LIN {X 0,Y 469.411,Z 470.46,A -85,B 0,C 180,E1 -7614.274,E2 -7614.274} C_VEL
LIN {X 0,Y 468.875,Z 476.006,A -85,B 0,C 180,E1 -7617.076,E2 -7617.076} C_VEL
LIN {X 0,Y 468.362,Z 482.236,A -85,B 0,C 180,E1 -7619.822,E2 -7619.822} C_VEL
LIN {X 0,Y 467.901,Z 490.724,A -85,B 0,C 180,E1 -7623.217,E2 -7623.217} C_VEL
LIN {X 0,Y 467.584,Z 498.381,A -85,B 0,C 180,E1 -7626.057,E2 -7626.057} C_VEL
LIN {X 0,Y 467.333,Z 507.548,A -85,B 0,C 180,E1 -7629.304,E2 -7629.304} C_VEL
LIN {X 0,Y 467.075,Z 516.898,A -85,B 0,C 180,E1 -7632.486,E2 -7632.486} C_VEL
LIN {X 0,Y 467.02,Z 523.224,A -85,B 0,C 180,E1 -7634.591,E2 -7634.591} C_VEL
LIN {X 0,Y 468.953,Z 538.487,A -85,B 0,C 180,E1 -7635.113,E2 -7635.113} C_VEL
LIN {X 0,Y 469.751,Z 545.686,A -85,B 0,C 180,E1 -7635.432,E2 -7635.432} C_VEL
LIN {X 0,Y 469.303,Z 557.555,A -85,B 0,C 180,E1 -7636.026,E2 -7636.026} C_VEL
LIN {X 0,Y 468.855,Z 569.316,A -85,B 0,C 180,E1 -7636.786,E2 -7636.786} C_VEL
LIN {X 0,Y 468.371,Z 580.525,A -85,B 0,C 180,E1 -7637.703,E2 -7637.703} C_VEL
LIN {X 0,Y 467.91,Z 590.813,A -85,B 0,C 180,E1 -7638.74,E2 -7638.74} C_VEL
LIN {X 0,Y 467.467,Z 599.647,A -85,B 0,C 180,E1 -7639.825,E2 -7639.825} C_VEL
LIN {X 0,Y 467.142,Z 608.26,A -85,B 0,C 180,E1 -7641.129,E2 -7641.129} C_VEL
LIN {X 0,Y 466.928,Z 615.206,A -85,B 0,C 180,E1 -7642.432,E2 -7642.432} C_VEL
LIN {X 0,Y 466.769,Z 621.589,A -85,B 0,C 180,E1 -7643.95,E2 -7643.95} C_VEL
LIN {X 0,Y 466.701,Z 625.734,A -85,B 0,C 180,E1 -7645.249,E2 -7645.249} C_VEL
LIN {X 0,Y 466.73,Z 628.807,A -85,B 0,C 180,E1 -7646.547,E2 -7646.547} C_VEL
LIN {X 0,Y 466.71,Z 630.278,A -85,B 0,C 180,E1 -7647.411,E2 -7647.411} C_VEL
LIN {X 0,Y 466.694,Z 631.332,A -85,B 0,C 180,E1 -7648.274,E2 -7648.274} C_VEL
LIN {X 0,Y 466.62,Z 631.982,A -85,B 0,C 180,E1 -7649.137,E2 -7649.137} C_VEL
LIN {X 0,Y 466.598,Z 632.228,A -85,B 0,C 180,E1 -7650,E2 -7650} C_VEL
LIN {X 0,Y 466.693,Z 631.43,A -85,B 0,C 180,E1 -7651.726,E2 -7651.726} C_VEL
LIN {X 0,Y 466.7,Z 630.431,A -85,B 0,C 180,E1 -7652.589,E2 -7652.589} C_VEL
LIN {X 0,Y 466.73,Z 629.01,A -85,B 0,C 180,E1 -7653.453,E2 -7653.453} C_VEL
LIN {X 0,Y 466.701,Z 626.022,A -85,B 0,C 180,E1 -7654.751,E2 -7654.751} C_VEL
LIN {X 0,Y 466.768,Z 621.97,A -85,B 0,C 180,E1 -7656.05,E2 -7656.05} C_VEL
LIN {X 0,Y 466.928,Z 615.723,A -85,B 0,C 180,E1 -7657.568,E2 -7657.568} C_VEL
LIN {X 0,Y 467.163,Z 608.913,A -85,B 0,C 180,E1 -7658.87,E2 -7658.87} C_VEL
LIN {X 0,Y 467.485,Z 600.458,A -85,B 0,C 180,E1 -7660.174,E2 -7660.174} C_VEL
LIN {X 0,Y 467.928,Z 591.764,A -85,B 0,C 180,E1 -7661.259,E2 -7661.259} C_VEL
LIN {X 0,Y 468.375,Z 581.539,A -85,B 0,C 180,E1 -7662.305,E2 -7662.305} C_VEL
LIN {X 0,Y 468.887,Z 570.553,A -85,B 0,C 180,E1 -7663.213,E2 -7663.213} C_VEL
LIN {X 0,Y 469.389,Z 558.907,A -85,B 0,C 180,E1 -7663.971,E2 -7663.971} C_VEL
LIN {X 0,Y 469.901,Z 545.767,A -85,B 0,C 180,E1 -7664.619,E2 -7664.619} C_VEL
LIN {X 0,Y 468.192,Z 532.419,A -85,B 0,C 180,E1 -7665.144,E2 -7665.144} C_VEL
LIN {X 0,Y 467.098,Z 524.822,A -85,B 0,C 180,E1 -7665.381,E2 -7665.381} C_VEL
LIN {X 0,Y 467.284,Z 515.355,A -85,B 0,C 180,E1 -7668.643,E2 -7668.643} C_VEL
LIN {X 0,Y 467.574,Z 505.589,A -85,B 0,C 180,E1 -7672.072,E2 -7672.072} C_VEL
LIN {X 0,Y 467.924,Z 496.629,A -85,B 0,C 180,E1 -7675.285,E2 -7675.285} C_VEL
LIN {X 0,Y 468.323,Z 488.674,A -85,B 0,C 180,E1 -7678.21,E2 -7678.21} C_VEL
LIN {X 0,Y 468.742,Z 480.586,A -85,B 0,C 180,E1 -7681.282,E2 -7681.282} C_VEL
LIN {X 0,Y 469.161,Z 473.387,A -85,B 0,C 180,E1 -7684.097,E2 -7684.097} C_VEL
LIN {X 0,Y 469.33,Z 468.592,A -85,B 0,C 180,E1 -7686.038,E2 -7686.038} C_VEL
LIN {X 0,Y 468.349,Z 462.399,A -85,B 0,C 180,E1 -7688.711,E2 -7688.711} C_VEL
LIN {X 0,Y 467.578,Z 458.244,A -85,B 0,C 180,E1 -7690.618,E2 -7690.618} C_VEL
LIN {X 0,Y 467.558,Z 458.244,A -85,B 0,C 180,E1 -7693.744,E2 -7693.744} C_VEL
LIN {X 0,Y 467.579,Z 458.244,A -85,B 0,C 180,E1 -7696.258,E2 -7696.258} C_VEL
LIN {X 0,Y 467.585,Z 458.241,A -85,B 0,C 180,E1 -7698.722,E2 -7698.722} C_VEL
LIN {X 0,Y 467.566,Z 458.242,A -85,B 0,C 180,E1 -7701.956,E2 -7701.956} C_VEL
LIN {X 0,Y 467.566,Z 458.245,A -85,B 0,C 180,E1 -7705.167,E2 -7705.167} C_VEL
LIN {X 0,Y 467.584,Z 458.241,A -85,B 0,C 180,E1 -7708.26,E2 -7708.26} C_VEL
LIN {X 0,Y 467.579,Z 458.243,A -85,B 0,C 180,E1 -7711.251,E2 -7711.251} C_VEL
LIN {X 0,Y 467.618,Z 458.238,A -85,B 0,C 180,E1 -7713.2,E2 -7713.2} C_VEL
LIN {X 0,Y 467.593,Z 458.243,A -85,B 0,C 180,E1 -7716.468,E2 -7716.468} C_VEL
LIN {X 0,Y 467.626,Z 458.236,A -85,B 0,C 180,E1 -7719.777,E2 -7719.777} C_VEL
LIN {X 0,Y 467.611,Z 458.24,A -85,B 0,C 180,E1 -7722.507,E2 -7722.507} C_VEL
LIN {X 0,Y 467.609,Z 458.238,A -85,B 0,C 180,E1 -7725.197,E2 -7725.197} C_VEL
LIN {X 0,Y 467.658,Z 458.232,A -85,B 0,C 180,E1 -7727.855,E2 -7727.855} C_VEL
LIN {X 0,Y 467.683,Z 458.228,A -85,B 0,C 180,E1 -7731.357,E2 -7731.357} C_VEL
LIN {X 0,Y 467.746,Z 458.222,A -85,B 0,C 180,E1 -7733.963,E2 -7733.963} C_VEL
LIN {X 0,Y 467.861,Z 458.204,A -85,B 0,C 180,E1 -7737.417,E2 -7737.417} C_VEL
LIN {X 0,Y 467.885,Z 458.206,A -85,B 0,C 180,E1 -7740,E2 -7740} C_VEL
LIN {X 0,Y 467.861,Z 458.208,A -85,B 0,C 180,E1 -7742.583,E2 -7742.583} C_VEL
LIN {X 0,Y 467.746,Z 458.223,A -85,B 0,C 180,E1 -7746.038,E2 -7746.038} C_VEL
LIN {X 0,Y 467.684,Z 458.229,A -85,B 0,C 180,E1 -7748.643,E2 -7748.643} C_VEL
LIN {X 0,Y 467.658,Z 458.233,A -85,B 0,C 180,E1 -7752.146,E2 -7752.146} C_VEL
LIN {X 0,Y 467.642,Z 458.235,A -85,B 0,C 180,E1 -7755.695,E2 -7755.695} C_VEL
LIN {X 0,Y 467.62,Z 458.236,A -85,B 0,C 180,E1 -7758.765,E2 -7758.765} C_VEL
LIN {X 0,Y 467.583,Z 458.241,A -85,B 0,C 180,E1 -7761.268,E2 -7761.268} C_VEL
LIN {X 0,Y 467.574,Z 458.242,A -85,B 0,C 180,E1 -7763.943,E2 -7763.943} C_VEL
LIN {X 0,Y 467.619,Z 458.236,A -85,B 0,C 180,E1 -7766.8,E2 -7766.8} C_VEL
LIN {X 0,Y 467.557,Z 458.246,A -85,B 0,C 180,E1 -7769.738,E2 -7769.738} C_VEL
LIN {X 0,Y 467.586,Z 458.24,A -85,B 0,C 180,E1 -7772.759,E2 -7772.759} C_VEL
LIN {X 0,Y 467.559,Z 458.247,A -85,B 0,C 180,E1 -7775.89,E2 -7775.89} C_VEL
LIN {X 0,Y 467.579,Z 458.241,A -85,B 0,C 180,E1 -7779.146,E2 -7779.146} C_VEL
LIN {X 0,Y 467.589,Z 458.24,A -85,B 0,C 180,E1 -7782.567,E2 -7782.567} C_VEL
LIN {X 0,Y 467.574,Z 458.243,A -85,B 0,C 180,E1 -7785.053,E2 -7785.053} C_VEL
LIN {X 0,Y 467.592,Z 458.238,A -85,B 0,C 180,E1 -7787.44,E2 -7787.44} C_VEL
LIN {X 0,Y 467.586,Z 458.242,A -85,B 0,C 180,E1 -7790.856,E2 -7790.856} C_VEL
LIN {X 0,Y 467.566,Z 458.246,A -85,B 0,C 180,E1 -7794.261,E2 -7794.261} C_VEL
LIN {X 0,Y 467.585,Z 458.241,A -85,B 0,C 180,E1 -7797.321,E2 -7797.321} C_VEL
LIN {X 0,Y 467.574,Z 458.243,A -85,B 0,C 180,E1 -7800.668,E2 -7800.668} C_VEL
LIN {X 0,Y 467.62,Z 458.235,A -85,B 0,C 180,E1 -7803.2,E2 -7803.2} C_VEL
LIN {X 0,Y 467.597,Z 458.241,A -85,B 0,C 180,E1 -7806.468,E2 -7806.468} C_VEL
LIN {X 0,Y 467.627,Z 458.236,A -85,B 0,C 180,E1 -7809.777,E2 -7809.777} C_VEL
LIN {X 0,Y 467.603,Z 458.239,A -85,B 0,C 180,E1 -7812.507,E2 -7812.507} C_VEL
LIN {X 0,Y 467.611,Z 458.237,A -85,B 0,C 180,E1 -7815.197,E2 -7815.197} C_VEL
LIN {X 0,Y 467.602,Z 458.238,A -85,B 0,C 180,E1 -7815.421,E2 -7815.421} C_VEL
LIN {X 0,Y 466.931,Z 458.326,A -85,B 0,C 180,E1 -7816.14,E2 -7816.14} C_VEL
LIN {X 0,Y 464.088,Z 458.675,A -85,B 0,C 180,E1 -7817.309,E2 -7817.309} C_VEL
LIN {X 0,Y 461.689,Z 458.975,A -85,B 0,C 180,E1 -7818.251,E2 -7818.251} C_VEL
LIN {X 0,Y 460.662,Z 459.103,A -85,B 0,C 180,E1 -7818.979,E2 -7818.979} C_VEL
LIN {X 0,Y 460.58,Z 459.113,A -85,B 0,C 180,E1 -7819.225,E2 -7819.225} C_VEL
LIN {X 0,Y 460.673,Z 459.102,A -85,B 0,C 180,E1 -7822.588,E2 -7822.588} C_VEL
LIN {X 0,Y 460.694,Z 459.098,A -85,B 0,C 180,E1 -7824.748,E2 -7824.748} C_VEL
LIN {X 0,Y 460.805,Z 459.087,A -85,B 0,C 180,E1 -7827.378,E2 -7827.378} C_VEL
LIN {X 0,Y 460.858,Z 459.081,A -85,B 0,C 180,E1 -7830,E2 -7830} C_VEL
LIN {X 0,Y 460.805,Z 459.084,A -85,B 0,C 180,E1 -7832.623,E2 -7832.623} C_VEL
LIN {X 0,Y 460.712,Z 459.099,A -85,B 0,C 180,E1 -7836.13,E2 -7836.13} C_VEL
LIN {X 0,Y 460.626,Z 459.106,A -85,B 0,C 180,E1 -7838.776,E2 -7838.776} C_VEL
LIN {X 0,Y 460.618,Z 459.111,A -85,B 0,C 180,E1 -7842.445,E2 -7842.445} C_VEL
LIN {X 0,Y 460.605,Z 459.112,A -85,B 0,C 180,E1 -7845.998,E2 -7845.998} C_VEL
LIN {X 0,Y 460.576,Z 459.114,A -85,B 0,C 180,E1 -7848.902,E2 -7848.902} C_VEL
LIN {X 0,Y 460.521,Z 459.12,A -85,B 0,C 180,E1 -7851.486,E2 -7851.486} C_VEL
LIN {X 0,Y 460.547,Z 459.117,A -85,B 0,C 180,E1 -7854.332,E2 -7854.332} C_VEL
LIN {X 0,Y 460.578,Z 459.114,A -85,B 0,C 180,E1 -7857.244,E2 -7857.244} C_VEL
LIN {X 0,Y 460.515,Z 459.121,A -85,B 0,C 180,E1 -7860.24,E2 -7860.24} C_VEL
LIN {X 0,Y 460.533,Z 459.121,A -85,B 0,C 180,E1 -7863.325,E2 -7863.325} C_VEL
LIN {X 0,Y 460.481,Z 459.124,A -85,B 0,C 180,E1 -7866.529,E2 -7866.529} C_VEL
LIN {X 0,Y 460.549,Z 459.117,A -85,B 0,C 180,E1 -7868.898,E2 -7868.898} C_VEL
LIN {X 0,Y 460.527,Z 459.122,A -85,B 0,C 180,E1 -7872.181,E2 -7872.181} C_VEL
LIN {X 0,Y 460.518,Z 459.122,A -85,B 0,C 180,E1 -7875.411,E2 -7875.411} C_VEL
LIN {X 0,Y 460.536,Z 459.12,A -85,B 0,C 180,E1 -7878.397,E2 -7878.397} C_VEL
LIN {X 0,Y 460.529,Z 459.119,A -85,B 0,C 180,E1 -7881.267,E2 -7881.267} C_VEL
LIN {X 0,Y 460.438,Z 459.132,A -85,B 0,C 180,E1 -7884.548,E2 -7884.548} C_VEL
LIN {X 0,Y 460.116,Z 459.175,A -85,B 0,C 180,E1 -7887.683,E2 -7887.683} C_VEL
LIN {X 0,Y 459.914,Z 459.335,A -85,B 0,C 180,E1 -7889.716,E2 -7889.716} C_VEL
LIN {X 0,Y 459.916,Z 462.429,A -85,B 0,C 180,E1 -7892.714,E2 -7892.714} C_VEL
LIN {X 0,Y 459.808,Z 465.5,A -85,B 0,C 180,E1 -7895.626,E2 -7895.626} C_VEL
LIN {X 0,Y 459.763,Z 468.905,A -85,B 0,C 180,E1 -7898.821,E2 -7898.821} C_VEL
LIN {X 0,Y 459.71,Z 472.578,A -85,B 0,C 180,E1 -7902.196,E2 -7902.196} C_VEL
LIN {X 0,Y 459.717,Z 475.164,A -85,B 0,C 180,E1 -7904.538,E2 -7904.538} C_VEL
LIN {X 0,Y 462.865,Z 489.688,A -85,B 0,C 180,E1 -7905.125,E2 -7905.125} C_VEL
LIN {X 0,Y 463.135,Z 494.215,A -85,B 0,C 180,E1 -7905.331,E2 -7905.331} C_VEL
LIN {X 0,Y 462.75,Z 505.895,A -85,B 0,C 180,E1 -7905.936,E2 -7905.936} C_VEL
LIN {X 0,Y 462.3,Z 517.223,A -85,B 0,C 180,E1 -7906.696,E2 -7906.696} C_VEL
LIN {X 0,Y 461.794,Z 528.968,A -85,B 0,C 180,E1 -7907.698,E2 -7907.698} C_VEL
LIN {X 0,Y 461.227,Z 539.33,A -85,B 0,C 180,E1 -7908.797,E2 -7908.797} C_VEL
LIN {X 0,Y 460.77,Z 549.23,A -85,B 0,C 180,E1 -7910.119,E2 -7910.119} C_VEL
LIN {X 0,Y 460.392,Z 557.21,A -85,B 0,C 180,E1 -7911.44,E2 -7911.44} C_VEL
LIN {X 0,Y 460.132,Z 562.609,A -85,B 0,C 180,E1 -7912.54,E2 -7912.54} C_VEL
LIN {X 0,Y 460.009,Z 567.893,A -85,B 0,C 180,E1 -7913.861,E2 -7913.861} C_VEL
LIN {X 0,Y 459.791,Z 572.006,A -85,B 0,C 180,E1 -7915.177,E2 -7915.177} C_VEL
LIN {X 0,Y 459.725,Z 575.053,A -85,B 0,C 180,E1 -7916.494,E2 -7916.494} C_VEL
LIN {X 0,Y 459.705,Z 576.536,A -85,B 0,C 180,E1 -7917.371,E2 -7917.371} C_VEL
LIN {X 0,Y 459.636,Z 577.592,A -85,B 0,C 180,E1 -7918.247,E2 -7918.247} C_VEL
LIN {X 0,Y 459.531,Z 578.546,A -85,B 0,C 180,E1 -7920,E2 -7920} C_VEL
LIN {X 0,Y 459.554,Z 578.388,A -85,B 0,C 180,E1 -7920.876,E2 -7920.876} C_VEL
LIN {X 0,Y 459.736,Z 576.871,A -85,B 0,C 180,E1 -7922.628,E2 -7922.628} C_VEL
LIN {X 0,Y 459.733,Z 575.522,A -85,B 0,C 180,E1 -7923.506,E2 -7923.506} C_VEL
LIN {X 0,Y 459.809,Z 572.652,A -85,B 0,C 180,E1 -7924.822,E2 -7924.822} C_VEL
LIN {X 0,Y 460.009,Z 568.73,A -85,B 0,C 180,E1 -7926.139,E2 -7926.139} C_VEL
LIN {X 0,Y 460.179,Z 563.651,A -85,B 0,C 180,E1 -7927.459,E2 -7927.459} C_VEL
LIN {X 0,Y 460.493,Z 557.247,A -85,B 0,C 180,E1 -7928.779,E2 -7928.779} C_VEL
LIN {X 0,Y 460.885,Z 549.276,A -85,B 0,C 180,E1 -7930.1,E2 -7930.1} C_VEL
LIN {X 0,Y 461.301,Z 541.139,A -85,B 0,C 180,E1 -7931.201,E2 -7931.201} C_VEL
LIN {X 0,Y 461.9,Z 531.186,A -85,B 0,C 180,E1 -7932.299,E2 -7932.299} C_VEL
LIN {X 0,Y 462.345,Z 519.856,A -85,B 0,C 180,E1 -7933.304,E2 -7933.304} C_VEL
LIN {X 0,Y 462.828,Z 509.159,A -85,B 0,C 180,E1 -7934.061,E2 -7934.061} C_VEL
LIN {X 0,Y 463.277,Z 497.241,A -85,B 0,C 180,E1 -7934.72,E2 -7934.72} C_VEL
LIN {X 0,Y 463.399,Z 492.393,A -85,B 0,C 180,E1 -7934.941,E2 -7934.941} C_VEL
LIN {X 0,Y 461.369,Z 482.734,A -85,B 0,C 180,E1 -7935.391,E2 -7935.391} C_VEL
LIN {X 0,Y 459.919,Z 477.276,A -85,B 0,C 180,E1 -7935.64,E2 -7935.64} C_VEL
LIN {X 0,Y 460.006,Z 474.424,A -85,B 0,C 180,E1 -7938.714,E2 -7938.714} C_VEL
LIN {X 0,Y 460.053,Z 471.957,A -85,B 0,C 180,E1 -7941.508,E2 -7941.508} C_VEL
LIN {X 0,Y 460.187,Z 469.59,A -85,B 0,C 180,E1 -7944.352,E2 -7944.352} C_VEL
LIN {X 0,Y 460.415,Z 466.954,A -85,B 0,C 180,E1 -7947.706,E2 -7947.706} C_VEL
LIN {X 0,Y 460.609,Z 464.479,A -85,B 0,C 180,E1 -7951.3,E2 -7951.3} C_VEL
LIN {X 0,Y 460.817,Z 462.698,A -85,B 0,C 180,E1 -7954.353,E2 -7954.353} C_VEL
LIN {X 0,Y 460.839,Z 461.746,A -85,B 0,C 180,E1 -7956.496,E2 -7956.496} C_VEL
LIN {X 0,Y 460.839,Z 461.064,A -85,B 0,C 180,E1 -7958.942,E2 -7958.942} C_VEL
LIN {X 0,Y 460.826,Z 460.856,A -85,B 0,C 180,E1 -7961.643,E2 -7961.643} C_VEL
LIN {X 0,Y 460.959,Z 461.487,A -85,B 0,C 180,E1 -7964.535,E2 -7964.535} C_VEL
LIN {X 0,Y 461.186,Z 462.915,A -85,B 0,C 180,E1 -7967.01,E2 -7967.01} C_VEL
LIN {X 0,Y 461.639,Z 465.205,A -85,B 0,C 180,E1 -7969.57,E2 -7969.57} C_VEL
LIN {X 0,Y 462.201,Z 468.615,A -85,B 0,C 180,E1 -7972.25,E2 -7972.25} C_VEL
LIN {X 0,Y 462.403,Z 470.846,A -85,B 0,C 180,E1 -7973.663,E2 -7973.663} C_VEL
LIN {X 0,Y 462.167,Z 474.66,A -85,B 0,C 180,E1 -7975.761,E2 -7975.761} C_VEL
LIN {X 0,Y 461.523,Z 481.094,A -85,B 0,C 180,E1 -7978.819,E2 -7978.819} C_VEL
LIN {X 0,Y 461.005,Z 489.008,A -85,B 0,C 180,E1 -7982.154,E2 -7982.154} C_VEL
LIN {X 0,Y 460.615,Z 496.842,A -85,B 0,C 180,E1 -7985.191,E2 -7985.191} C_VEL
LIN {X 0,Y 460.323,Z 505.906,A -85,B 0,C 180,E1 -7988.505,E2 -7988.505} C_VEL
LIN {X 0,Y 460.059,Z 515.164,A -85,B 0,C 180,E1 -7991.75,E2 -7991.75} C_VEL
LIN {X 0,Y 459.944,Z 522.743,A -85,B 0,C 180,E1 -7994.336,E2 -7994.336} C_VEL
LIN {X 0,Y 461.694,Z 536.071,A -85,B 0,C 180,E1 -7994.79,E2 -7994.79} C_VEL
LIN {X 0,Y 462.832,Z 546.609,A -85,B 0,C 180,E1 -7995.265,E2 -7995.265} C_VEL
LIN {X 0,Y 462.324,Z 559.032,A -85,B 0,C 180,E1 -7995.923,E2 -7995.923} C_VEL
LIN {X 0,Y 461.735,Z 571.691,A -85,B 0,C 180,E1 -7996.802,E2 -7996.802} C_VEL
LIN {X 0,Y 461.195,Z 583.009,A -85,B 0,C 180,E1 -7997.793,E2 -7997.793} C_VEL
LIN {X 0,Y 460.783,Z 592.205,A -85,B 0,C 180,E1 -7998.786,E2 -7998.786} C_VEL
LIN {X 0,Y 460.297,Z 602.22,A -85,B 0,C 180,E1 -8000.109,E2 -8000.109} C_VEL
LIN {X 0,Y 460.03,Z 610.282,A -85,B 0,C 180,E1 -8001.434,E2 -8001.434} C_VEL
LIN {X 0,Y 459.775,Z 617.67,A -85,B 0,C 180,E1 -8002.976,E2 -8002.976} C_VEL
LIN {X 0,Y 459.683,Z 622.616,A -85,B 0,C 180,E1 -8004.297,E2 -8004.297} C_VEL
LIN {X 0,Y 459.587,Z 626.407,A -85,B 0,C 180,E1 -8005.615,E2 -8005.615} C_VEL
LIN {X 0,Y 459.643,Z 628.375,A -85,B 0,C 180,E1 -8006.493,E2 -8006.493} C_VEL
LIN {X 0,Y 459.63,Z 629.853,A -85,B 0,C 180,E1 -8007.371,E2 -8007.371} C_VEL
LIN {X 0,Y 459.631,Z 630.914,A -85,B 0,C 180,E1 -8008.247,E2 -8008.247} C_VEL
LIN {X 0,Y 459.553,Z 631.57,A -85,B 0,C 180,E1 -8009.124,E2 -8009.124} C_VEL
LIN {X 0,Y 459.53,Z 631.819,A -85,B 0,C 180,E1 -8010,E2 -8010} C_VEL
LIN {X 0,Y 459.553,Z 631.62,A -85,B 0,C 180,E1 -8010.876,E2 -8010.876} C_VEL
LIN {X 0,Y 459.63,Z 631.024,A -85,B 0,C 180,E1 -8011.752,E2 -8011.752} C_VEL
LIN {X 0,Y 459.621,Z 630.022,A -85,B 0,C 180,E1 -8012.629,E2 -8012.629} C_VEL
LIN {X 0,Y 459.627,Z 628.595,A -85,B 0,C 180,E1 -8013.506,E2 -8013.506} C_VEL
LIN {X 0,Y 459.631,Z 625.603,A -85,B 0,C 180,E1 -8014.824,E2 -8014.824} C_VEL
LIN {X 0,Y 459.714,Z 620.477,A -85,B 0,C 180,E1 -8016.431,E2 -8016.431} C_VEL
LIN {X 0,Y 459.896,Z 614.255,A -85,B 0,C 180,E1 -8017.905,E2 -8017.905} C_VEL
LIN {X 0,Y 460.185,Z 607.179,A -85,B 0,C 180,E1 -8019.228,E2 -8019.228} C_VEL
LIN {X 0,Y 460.537,Z 598.326,A -85,B 0,C 180,E1 -8020.552,E2 -8020.552} C_VEL
LIN {X 0,Y 461.115,Z 588.309,A -85,B 0,C 180,E1 -8021.762,E2 -8021.762} C_VEL
LIN {X 0,Y 461.583,Z 578.318,A -85,B 0,C 180,E1 -8022.736,E2 -8022.736} C_VEL
LIN {X 0,Y 462.104,Z 566.89,A -85,B 0,C 180,E1 -8023.635,E2 -8023.635} C_VEL
LIN {X 0,Y 462.627,Z 554.388,A -85,B 0,C 180,E1 -8024.404,E2 -8024.404} C_VEL
LIN {X 0,Y 462.869,Z 545.124,A -85,B 0,C 180,E1 -8024.846,E2 -8024.846} C_VEL
LIN {X 0,Y 461.093,Z 531.876,A -85,B 0,C 180,E1 -8025.378,E2 -8025.378} C_VEL
LIN {X 0,Y 460.036,Z 524.518,A -85,B 0,C 180,E1 -8025.612,E2 -8025.612} C_VEL
LIN {X 0,Y 460.245,Z 514.537,A -85,B 0,C 180,E1 -8029.12,E2 -8029.12} C_VEL
LIN {X 0,Y 460.516,Z 505.288,A -85,B 0,C 180,E1 -8032.428,E2 -8032.428} C_VEL
LIN {X 0,Y 460.864,Z 497.511,A -85,B 0,C 180,E1 -8035.277,E2 -8035.277} C_VEL
LIN {X 0,Y 461.294,Z 489.756,A -85,B 0,C 180,E1 -8038.184,E2 -8038.184} C_VEL
LIN {X 0,Y 461.739,Z 481.06,A -85,B 0,C 180,E1 -8041.53,E2 -8041.53} C_VEL
LIN {X 0,Y 462.177,Z 474.275,A -85,B 0,C 180,E1 -8044.238,E2 -8044.238} C_VEL
LIN {X 0,Y 462.254,Z 469.238,A -85,B 0,C 180,E1 -8046.312,E2 -8046.312} C_VEL
LIN {X 0,Y 461.283,Z 463.124,A -85,B 0,C 180,E1 -8049.011,E2 -8049.011} C_VEL
LIN {X 0,Y 460.549,Z 459.12,A -85,B 0,C 180,E1 -8050.912,E2 -8050.912} C_VEL
LIN {X 0,Y 460.513,Z 459.123,A -85,B 0,C 180,E1 -8054.17,E2 -8054.17} C_VEL
LIN {X 0,Y 460.544,Z 459.118,A -85,B 0,C 180,E1 -8057.096,E2 -8057.096} C_VEL
LIN {X 0,Y 460.529,Z 459.118,A -85,B 0,C 180,E1 -8060.137,E2 -8060.137} C_VEL
LIN {X 0,Y 460.478,Z 459.127,A -85,B 0,C 180,E1 -8063.471,E2 -8063.471} C_VEL
LIN {X 0,Y 460.53,Z 459.121,A -85,B 0,C 180,E1 -8066.675,E2 -8066.675} C_VEL
LIN {X 0,Y 460.512,Z 459.121,A -85,B 0,C 180,E1 -8069.76,E2 -8069.76} C_VEL
LIN {X 0,Y 460.581,Z 459.114,A -85,B 0,C 180,E1 -8072.757,E2 -8072.757} C_VEL
LIN {X 0,Y 460.542,Z 459.116,A -85,B 0,C 180,E1 -8075.668,E2 -8075.668} C_VEL
LIN {X 0,Y 460.523,Z 459.121,A -85,B 0,C 180,E1 -8078.578,E2 -8078.578} C_VEL
LIN {X 0,Y 460.593,Z 459.111,A -85,B 0,C 180,E1 -8081.311,E2 -8081.311} C_VEL
LIN {X 0,Y 460.606,Z 459.111,A -85,B 0,C 180,E1 -8084.059,E2 -8084.059} C_VEL
LIN {X 0,Y 460.611,Z 459.11,A -85,B 0,C 180,E1 -8087.666,E2 -8087.666} C_VEL
LIN {X 0,Y 460.63,Z 459.106,A -85,B 0,C 180,E1 -8091.224,E2 -8091.224} C_VEL
LIN {X 0,Y 460.712,Z 459.098,A -85,B 0,C 180,E1 -8093.87,E2 -8093.87} C_VEL
LIN {X 0,Y 460.802,Z 459.083,A -85,B 0,C 180,E1 -8097.378,E2 -8097.378} C_VEL
LIN {X 0,Y 460.856,Z 459.081,A -85,B 0,C 180,E1 -8100,E2 -8100} C_VEL
LIN {X 0,Y 460.826,Z 459.085,A -85,B 0,C 180,E1 -8102.623,E2 -8102.623} C_VEL
LIN {X 0,Y 460.712,Z 459.1,A -85,B 0,C 180,E1 -8106.13,E2 -8106.13} C_VEL
LIN {X 0,Y 460.631,Z 459.109,A -85,B 0,C 180,E1 -8108.776,E2 -8108.776} C_VEL
LIN {X 0,Y 460.616,Z 459.111,A -85,B 0,C 180,E1 -8112.445,E2 -8112.445} C_VEL
LIN {X 0,Y 460.602,Z 459.111,A -85,B 0,C 180,E1 -8115.998,E2 -8115.998} C_VEL
LIN {X 0,Y 460.574,Z 459.113,A -85,B 0,C 180,E1 -8118.902,E2 -8118.902} C_VEL
LIN {X 0,Y 460.518,Z 459.121,A -85,B 0,C 180,E1 -8121.486,E2 -8121.486} C_VEL
LIN {X 0,Y 460.544,Z 459.119,A -85,B 0,C 180,E1 -8124.332,E2 -8124.332} C_VEL
LIN {X 0,Y 460.582,Z 459.112,A -85,B 0,C 180,E1 -8127.244,E2 -8127.244} C_VEL
LIN {X 0,Y 460.514,Z 459.122,A -85,B 0,C 180,E1 -8130.24,E2 -8130.24} C_VEL
LIN {X 0,Y 460.532,Z 459.116,A -85,B 0,C 180,E1 -8133.325,E2 -8133.325} C_VEL
LIN {X 0,Y 460.482,Z 459.126,A -85,B 0,C 180,E1 -8136.529,E2 -8136.529} C_VEL
LIN {X 0,Y 460.544,Z 459.118,A -85,B 0,C 180,E1 -8138.897,E2 -8138.897} C_VEL
LIN {X 0,Y 460.527,Z 459.122,A -85,B 0,C 180,E1 -8142.181,E2 -8142.181} C_VEL
LIN {X 0,Y 460.52,Z 459.121,A -85,B 0,C 180,E1 -8145.412,E2 -8145.412} C_VEL
LIN {X 0,Y 460.535,Z 459.12,A -85,B 0,C 180,E1 -8148.398,E2 -8148.398} C_VEL
LIN {X 0,Y 460.53,Z 459.12,A -85,B 0,C 180,E1 -8151.267,E2 -8151.267} C_VEL
LIN {X 0,Y 460.517,Z 459.122,A -85,B 0,C 180,E1 -8154.555,E2 -8154.555} C_VEL
LIN {X 0,Y 460.535,Z 459.121,A -85,B 0,C 180,E1 -8157.716,E2 -8157.716} C_VEL
LIN {X 0,Y 460.544,Z 459.118,A -85,B 0,C 180,E1 -8160.769,E2 -8160.769} C_VEL
LIN {X 0,Y 460.567,Z 459.117,A -85,B 0,C 180,E1 -8163.735,E2 -8163.735} C_VEL
LIN {X 0,Y 460.55,Z 459.119,A -85,B 0,C 180,E1 -8166.624,E2 -8166.624} C_VEL
LIN {X 0,Y 460.555,Z 459.115,A -85,B 0,C 180,E1 -8169.453,E2 -8169.453} C_VEL
LIN {X 0,Y 460.554,Z 459.117,A -85,B 0,C 180,E1 -8172.23,E2 -8172.23} C_VEL
LIN {X 0,Y 460.57,Z 459.114,A -85,B 0,C 180,E1 -8174.965,E2 -8174.965} C_VEL
LIN {X 0,Y 460.616,Z 459.108,A -85,B 0,C 180,E1 -8178.559,E2 -8178.559} C_VEL
LIN {X 0,Y 460.58,Z 459.113,A -85,B 0,C 180,E1 -8179.225,E2 -8179.225} C_VEL
LIN {X 0,Y 459.918,Z 459.199,A -85,B 0,C 180,E1 -8179.955,E2 -8179.955} C_VEL
LIN {X 0,Y 457.076,Z 459.553,A -85,B 0,C 180,E1 -8181.141,E2 -8181.141} C_VEL
LIN {X 0,Y 454.683,Z 459.849,A -85,B 0,C 180,E1 -8182.098,E2 -8182.098} C_VEL
LIN {X 0,Y 453.672,Z 459.973,A -85,B 0,C 180,E1 -8182.837,E2 -8182.837} C_VEL
LIN {X 0,Y 453.599,Z 459.981,A -85,B 0,C 180,E1 -8183.087,E2 -8183.087} C_VEL
LIN {X 0,Y 453.667,Z 459.973,A -85,B 0,C 180,E1 -8184.667,E2 -8184.667} C_VEL
LIN {X 0,Y 453.749,Z 459.965,A -85,B 0,C 180,E1 -8187.337,E2 -8187.337} C_VEL
LIN {X 0,Y 453.828,Z 459.956,A -85,B 0,C 180,E1 -8190,E2 -8190} C_VEL
LIN {X 0,Y 453.749,Z 459.964,A -85,B 0,C 180,E1 -8192.663,E2 -8192.663} C_VEL
LIN {X 0,Y 453.678,Z 459.976,A -85,B 0,C 180,E1 -8196.225,E2 -8196.225} C_VEL
LIN {X 0,Y 453.591,Z 459.982,A -85,B 0,C 180,E1 -8198.914,E2 -8198.914} C_VEL
LIN {X 0,Y 453.568,Z 459.988,A -85,B 0,C 180,E1 -8202.529,E2 -8202.529} C_VEL
LIN {X 0,Y 453.55,Z 459.989,A -85,B 0,C 180,E1 -8206.196,E2 -8206.196} C_VEL
LIN {X 0,Y 453.525,Z 459.992,A -85,B 0,C 180,E1 -8209.041,E2 -8209.041} C_VEL
LIN {X 0,Y 453.481,Z 459.999,A -85,B 0,C 180,E1 -8211.836,E2 -8211.836} C_VEL
LIN {X 0,Y 453.518,Z 459.993,A -85,B 0,C 180,E1 -8214.734,E2 -8214.734} C_VEL
LIN {X 0,Y 453.537,Z 459.992,A -85,B 0,C 180,E1 -8217.96,E2 -8217.96} C_VEL
LIN {X 0,Y 453.471,Z 460.001,A -85,B 0,C 180,E1 -8221.525,E2 -8221.525} C_VEL
LIN {X 0,Y 453.492,Z 459.996,A -85,B 0,C 180,E1 -8224.777,E2 -8224.777} C_VEL
LIN {X 0,Y 453.477,Z 459.997,A -85,B 0,C 180,E1 -8228.311,E2 -8228.311} C_VEL
LIN {X 0,Y 453.498,Z 459.996,A -85,B 0,C 180,E1 -8230.609,E2 -8230.609} C_VEL
LIN {X 0,Y 453.458,Z 460,A -85,B 0,C 180,E1 -8233.244,E2 -8233.244} C_VEL
LIN {X 0,Y 453.468,Z 460.001,A -85,B 0,C 180,E1 -8235.779,E2 -8235.779} C_VEL
LIN {X 0,Y 453.483,Z 459.999,A -85,B 0,C 180,E1 -8238.209,E2 -8238.209} C_VEL
LIN {X 0,Y 453.497,Z 459.994,A -85,B 0,C 180,E1 -8240.793,E2 -8240.793} C_VEL
LIN {X 0,Y 453.416,Z 460.006,A -85,B 0,C 180,E1 -8243.913,E2 -8243.913} C_VEL
LIN {X 0,Y 453.264,Z 460.028,A -85,B 0,C 180,E1 -8246.069,E2 -8246.069} C_VEL
LIN {X 0,Y 452.902,Z 460.073,A -85,B 0,C 180,E1 -8249.197,E2 -8249.197} C_VEL
LIN {X 0,Y 452.825,Z 460.665,A -85,B 0,C 180,E1 -8250.359,E2 -8250.359} C_VEL
LIN {X 0,Y 452.802,Z 463.637,A -85,B 0,C 180,E1 -8253.249,E2 -8253.249} C_VEL
LIN {X 0,Y 452.713,Z 466.879,A -85,B 0,C 180,E1 -8256.338,E2 -8256.338} C_VEL
LIN {X 0,Y 452.689,Z 469.796,A -85,B 0,C 180,E1 -8259.079,E2 -8259.079} C_VEL
LIN {X 0,Y 452.659,Z 472.859,A -85,B 0,C 180,E1 -8261.909,E2 -8261.909} C_VEL
LIN {X 0,Y 452.634,Z 475.482,A -85,B 0,C 180,E1 -8264.296,E2 -8264.296} C_VEL
LIN {X 0,Y 455.941,Z 490.334,A -85,B 0,C 180,E1 -8264.923,E2 -8264.923} C_VEL
LIN {X 0,Y 456.263,Z 494.185,A -85,B 0,C 180,E1 -8265.105,E2 -8265.105} C_VEL
LIN {X 0,Y 455.869,Z 505.927,A -85,B 0,C 180,E1 -8265.719,E2 -8265.719} C_VEL
LIN {X 0,Y 455.382,Z 517.236,A -85,B 0,C 180,E1 -8266.482,E2 -8266.482} C_VEL
LIN {X 0,Y 454.851,Z 529.115,A -85,B 0,C 180,E1 -8267.507,E2 -8267.507} C_VEL
LIN {X 0,Y 454.264,Z 539.526,A -85,B 0,C 180,E1 -8268.623,E2 -8268.623} C_VEL
LIN {X 0,Y 453.782,Z 549.467,A -85,B 0,C 180,E1 -8269.966,E2 -8269.966} C_VEL
LIN {X 0,Y 453.364,Z 557.483,A -85,B 0,C 180,E1 -8271.307,E2 -8271.307} C_VEL
LIN {X 0,Y 453.078,Z 562.908,A -85,B 0,C 180,E1 -8272.423,E2 -8272.423} C_VEL
LIN {X 0,Y 452.972,Z 568.218,A -85,B 0,C 180,E1 -8273.765,E2 -8273.765} C_VEL
LIN {X 0,Y 452.705,Z 572.359,A -85,B 0,C 180,E1 -8275.102,E2 -8275.102} C_VEL
LIN {X 0,Y 452.667,Z 575.425,A -85,B 0,C 180,E1 -8276.439,E2 -8276.439} C_VEL
LIN {X 0,Y 452.624,Z 576.924,A -85,B 0,C 180,E1 -8277.33,E2 -8277.33} C_VEL
LIN {X 0,Y 452.577,Z 577.991,A -85,B 0,C 180,E1 -8278.22,E2 -8278.22} C_VEL
LIN {X 0,Y 452.465,Z 578.96,A -85,B 0,C 180,E1 -8280,E2 -8280} C_VEL
LIN {X 0,Y 452.49,Z 578.809,A -85,B 0,C 180,E1 -8280.89,E2 -8280.89} C_VEL
LIN {X 0,Y 452.579,Z 578.25,A -85,B 0,C 180,E1 -8281.78,E2 -8281.78} C_VEL
LIN {X 0,Y 452.652,Z 577.303,A -85,B 0,C 180,E1 -8282.67,E2 -8282.67} C_VEL
LIN {X 0,Y 452.676,Z 575.96,A -85,B 0,C 180,E1 -8283.56,E2 -8283.56} C_VEL
LIN {X 0,Y 452.74,Z 573.105,A -85,B 0,C 180,E1 -8284.898,E2 -8284.898} C_VEL
LIN {X 0,Y 453.028,Z 568.123,A -85,B 0,C 180,E1 -8286.541,E2 -8286.541} C_VEL
LIN {X 0,Y 453.244,Z 562.162,A -85,B 0,C 180,E1 -8288.022,E2 -8288.022} C_VEL
LIN {X 0,Y 453.657,Z 555.311,A -85,B 0,C 180,E1 -8289.361,E2 -8289.361} C_VEL
LIN {X 0,Y 454.099,Z 546.715,A -85,B 0,C 180,E1 -8290.703,E2 -8290.703} C_VEL
LIN {X 0,Y 454.562,Z 537.924,A -85,B 0,C 180,E1 -8291.821,E2 -8291.821} C_VEL
LIN {X 0,Y 455.224,Z 527.276,A -85,B 0,C 180,E1 -8292.918,E2 -8292.918} C_VEL
LIN {X 0,Y 455.684,Z 516.288,A -85,B 0,C 180,E1 -8293.83,E2 -8293.83} C_VEL
LIN {X 0,Y 456.24,Z 503.452,A -85,B 0,C 180,E1 -8294.667,E2 -8294.667} C_VEL
LIN {X 0,Y 456.601,Z 493.437,A -85,B 0,C 180,E1 -8295.169,E2 -8295.169} C_VEL
LIN {X 0,Y 454.459,Z 483.598,A -85,B 0,C 180,E1 -8295.65,E2 -8295.65} C_VEL
LIN {X 0,Y 452.898,Z 477.864,A -85,B 0,C 180,E1 -8295.908,E2 -8295.908} C_VEL
LIN {X 0,Y 452.958,Z 475.034,A -85,B 0,C 180,E1 -8299.016,E2 -8299.016} C_VEL
LIN {X 0,Y 453.018,Z 472.586,A -85,B 0,C 180,E1 -8301.859,E2 -8301.859} C_VEL
LIN {X 0,Y 453.174,Z 470.243,A -85,B 0,C 180,E1 -8304.754,E2 -8304.754} C_VEL
LIN {X 0,Y 453.412,Z 467.846,A -85,B 0,C 180,E1 -8307.93,E2 -8307.93} C_VEL
LIN {X 0,Y 453.61,Z 465.473,A -85,B 0,C 180,E1 -8311.554,E2 -8311.554} C_VEL
LIN {X 0,Y 453.783,Z 464.18,A -85,B 0,C 180,E1 -8313.887,E2 -8313.887} C_VEL
LIN {X 0,Y 453.873,Z 463.111,A -85,B 0,C 180,E1 -8316.371,E2 -8316.371} C_VEL
LIN {X 0,Y 453.851,Z 462.372,A -85,B 0,C 180,E1 -8319.412,E2 -8319.412} C_VEL
LIN {X 0,Y 453.898,Z 462.386,A -85,B 0,C 180,E1 -8321.994,E2 -8321.994} C_VEL
LIN {X 0,Y 454.032,Z 463.075,A -85,B 0,C 180,E1 -8324.599,E2 -8324.599} C_VEL
LIN {X 0,Y 454.275,Z 464.557,A -85,B 0,C 180,E1 -8327.1,E2 -8327.1} C_VEL
LIN {X 0,Y 454.709,Z 466.748,A -85,B 0,C 180,E1 -8329.522,E2 -8329.522} C_VEL
LIN {X 0,Y 455.205,Z 469.702,A -85,B 0,C 180,E1 -8331.943,E2 -8331.943} C_VEL
LIN {X 0,Y 455.395,Z 473.018,A -85,B 0,C 180,E1 -8334.095,E2 -8334.095} C_VEL
LIN {X 0,Y 455.038,Z 477.48,A -85,B 0,C 180,E1 -8336.514,E2 -8336.514} C_VEL
LIN {X 0,Y 454.442,Z 483.397,A -85,B 0,C 180,E1 -8339.313,E2 -8339.313} C_VEL
LIN {X 0,Y 453.87,Z 491.671,A -85,B 0,C 180,E1 -8342.819,E2 -8342.819} C_VEL
LIN {X 0,Y 453.491,Z 499.158,A -85,B 0,C 180,E1 -8345.745,E2 -8345.745} C_VEL
LIN {X 0,Y 453.212,Z 508.197,A -85,B 0,C 180,E1 -8349.104,E2 -8349.104} C_VEL
LIN {X 0,Y 452.935,Z 517.436,A -85,B 0,C 180,E1 -8352.388,E2 -8352.388} C_VEL
LIN {X 0,Y 452.884,Z 522.462,A -85,B 0,C 180,E1 -8354.059,E2 -8354.059} C_VEL
LIN {X 0,Y 454.645,Z 535.205,A -85,B 0,C 180,E1 -8354.512,E2 -8354.512} C_VEL
LIN {X 0,Y 455.916,Z 547.658,A -85,B 0,C 180,E1 -8355.094,E2 -8355.094} C_VEL
LIN {X 0,Y 455.323,Z 560.449,A -85,B 0,C 180,E1 -8355.816,E2 -8355.816} C_VEL
LIN {X 0,Y 454.705,Z 573.17,A -85,B 0,C 180,E1 -8356.747,E2 -8356.747} C_VEL
LIN {X 0,Y 454.151,Z 583.647,A -85,B 0,C 180,E1 -8357.714,E2 -8357.714} C_VEL
LIN {X 0,Y 453.699,Z 593.572,A -85,B 0,C 180,E1 -8358.835,E2 -8358.835} C_VEL
LIN {X 0,Y 453.26,Z 601.76,A -85,B 0,C 180,E1 -8359.954,E2 -8359.954} C_VEL
LIN {X 0,Y 452.962,Z 609.819,A -85,B 0,C 180,E1 -8361.299,E2 -8361.299} C_VEL
LIN {X 0,Y 452.757,Z 615.313,A -85,B 0,C 180,E1 -8362.418,E2 -8362.418} C_VEL
LIN {X 0,Y 452.604,Z 620.68,A -85,B 0,C 180,E1 -8363.76,E2 -8363.76} C_VEL
LIN {X 0,Y 452.562,Z 624.855,A -85,B 0,C 180,E1 -8365.1,E2 -8365.1} C_VEL
LIN {X 0,Y 452.542,Z 627.948,A -85,B 0,C 180,E1 -8366.438,E2 -8366.438} C_VEL
LIN {X 0,Y 452.552,Z 629.433,A -85,B 0,C 180,E1 -8367.33,E2 -8367.33} C_VEL
LIN {X 0,Y 452.539,Z 630.498,A -85,B 0,C 180,E1 -8368.22,E2 -8368.22} C_VEL
LIN {X 0,Y 452.489,Z 631.158,A -85,B 0,C 180,E1 -8369.11,E2 -8369.11} C_VEL
LIN {X 0,Y 452.463,Z 631.408,A -85,B 0,C 180,E1 -8370,E2 -8370} C_VEL
LIN {X 0,Y 452.489,Z 631.21,A -85,B 0,C 180,E1 -8370.89,E2 -8370.89} C_VEL
LIN {X 0,Y 452.538,Z 630.612,A -85,B 0,C 180,E1 -8371.78,E2 -8371.78} C_VEL
LIN {X 0,Y 452.543,Z 629.61,A -85,B 0,C 180,E1 -8372.67,E2 -8372.67} C_VEL
LIN {X 0,Y 452.527,Z 628.175,A -85,B 0,C 180,E1 -8373.562,E2 -8373.562} C_VEL
LIN {X 0,Y 452.561,Z 625.177,A -85,B 0,C 180,E1 -8374.9,E2 -8374.9} C_VEL
LIN {X 0,Y 452.61,Z 620.532,A -85,B 0,C 180,E1 -8376.396,E2 -8376.396} C_VEL
LIN {X 0,Y 452.843,Z 613.796,A -85,B 0,C 180,E1 -8378.029,E2 -8378.029} C_VEL
LIN {X 0,Y 453.121,Z 606.687,A -85,B 0,C 180,E1 -8379.373,E2 -8379.373} C_VEL
LIN {X 0,Y 453.523,Z 597.81,A -85,B 0,C 180,E1 -8380.717,E2 -8380.717} C_VEL
LIN {X 0,Y 454.099,Z 587.755,A -85,B 0,C 180,E1 -8381.947,E2 -8381.947} C_VEL
LIN {X 0,Y 454.617,Z 577.523,A -85,B 0,C 180,E1 -8382.953,E2 -8382.953} C_VEL
LIN {X 0,Y 455.16,Z 566.255,A -85,B 0,C 180,E1 -8383.847,E2 -8383.847} C_VEL
LIN {X 0,Y 455.628,Z 555.675,A -85,B 0,C 180,E1 -8384.516,E2 -8384.516} C_VEL
LIN {X 0,Y 455.869,Z 545.616,A -85,B 0,C 180,E1 -8385.022,E2 -8385.022} C_VEL
LIN {X 0,Y 454.12,Z 532.212,A -85,B 0,C 180,E1 -8385.582,E2 -8385.582} C_VEL
LIN {X 0,Y 452.928,Z 524.229,A -85,B 0,C 180,E1 -8385.836,E2 -8385.836} C_VEL
LIN {X 0,Y 453.156,Z 515.37,A -85,B 0,C 180,E1 -8389.007,E2 -8389.007} C_VEL
LIN {X 0,Y 453.454,Z 506.291,A -85,B 0,C 180,E1 -8392.316,E2 -8392.316} C_VEL
LIN {X 0,Y 453.801,Z 498.543,A -85,B 0,C 180,E1 -8395.207,E2 -8395.207} C_VEL
LIN {X 0,Y 454.315,Z 489.484,A -85,B 0,C 180,E1 -8398.656,E2 -8398.656} C_VEL
LIN {X 0,Y 454.875,Z 480.478,A -85,B 0,C 180,E1 -8402.212,E2 -8402.212} C_VEL
LIN {X 0,Y 455.298,Z 473.384,A -85,B 0,C 180,E1 -8405.104,E2 -8405.104} C_VEL
LIN {X 0,Y 455.212,Z 469.866,A -85,B 0,C 180,E1 -8406.599,E2 -8406.599} C_VEL
LIN {X 0,Y 454.18,Z 463.697,A -85,B 0,C 180,E1 -8409.378,E2 -8409.378} C_VEL
LIN {X 0,Y 453.502,Z 459.998,A -85,B 0,C 180,E1 -8411.195,E2 -8411.195} C_VEL
LIN {X 0,Y 453.489,Z 459.999,A -85,B 0,C 180,E1 -8414.529,E2 -8414.529} C_VEL
LIN {X 0,Y 453.496,Z 459.997,A -85,B 0,C 180,E1 -8418.063,E2 -8418.063} C_VEL
LIN {X 0,Y 453.492,Z 459.999,A -85,B 0,C 180,E1 -8420.794,E2 -8420.794} C_VEL
LIN {X 0,Y 453.455,Z 460.001,A -85,B 0,C 180,E1 -8423.917,E2 -8423.917} C_VEL
LIN {X 0,Y 453.484,Z 459.998,A -85,B 0,C 180,E1 -8427.151,E2 -8427.151} C_VEL
LIN {X 0,Y 453.477,Z 460,A -85,B 0,C 180,E1 -8430.268,E2 -8430.268} C_VEL
LIN {X 0,Y 453.511,Z 459.994,A -85,B 0,C 180,E1 -8433.294,E2 -8433.294} C_VEL
LIN {X 0,Y 453.503,Z 459.995,A -85,B 0,C 180,E1 -8436.239,E2 -8436.239} C_VEL
LIN {X 0,Y 453.485,Z 459.999,A -85,B 0,C 180,E1 -8439.118,E2 -8439.118} C_VEL
LIN {X 0,Y 453.514,Z 459.992,A -85,B 0,C 180,E1 -8441.945,E2 -8441.945} C_VEL
LIN {X 0,Y 453.542,Z 459.99,A -85,B 0,C 180,E1 -8444.726,E2 -8444.726} C_VEL
LIN {X 0,Y 453.562,Z 459.988,A -85,B 0,C 180,E1 -8448.379,E2 -8448.379} C_VEL
LIN {X 0,Y 453.654,Z 459.977,A -85,B 0,C 180,E1 -8451.985,E2 -8451.985} C_VEL
LIN {X 0,Y 453.673,Z 459.975,A -85,B 0,C 180,E1 -8454.667,E2 -8454.667} C_VEL
LIN {X 0,Y 453.746,Z 459.962,A -85,B 0,C 180,E1 -8457.337,E2 -8457.337} C_VEL
LIN {X 0,Y 453.826,Z 459.957,A -85,B 0,C 180,E1 -8460,E2 -8460} C_VEL
LIN {X 0,Y 453.766,Z 459.965,A -85,B 0,C 180,E1 -8462.663,E2 -8462.663} C_VEL
LIN {X 0,Y 453.68,Z 459.976,A -85,B 0,C 180,E1 -8466.225,E2 -8466.225} C_VEL
LIN {X 0,Y 453.595,Z 459.986,A -85,B 0,C 180,E1 -8468.914,E2 -8468.914} C_VEL
LIN {X 0,Y 453.566,Z 459.988,A -85,B 0,C 180,E1 -8472.529,E2 -8472.529} C_VEL
LIN {X 0,Y 453.547,Z 459.99,A -85,B 0,C 180,E1 -8476.196,E2 -8476.196} C_VEL
LIN {X 0,Y 453.523,Z 459.991,A -85,B 0,C 180,E1 -8479.041,E2 -8479.041} C_VEL
LIN {X 0,Y 453.479,Z 460,A -85,B 0,C 180,E1 -8481.836,E2 -8481.836} C_VEL
LIN {X 0,Y 453.516,Z 459.995,A -85,B 0,C 180,E1 -8484.735,E2 -8484.735} C_VEL
LIN {X 0,Y 453.54,Z 459.992,A -85,B 0,C 180,E1 -8487.961,E2 -8487.961} C_VEL
LIN {X 0,Y 453.469,Z 459.999,A -85,B 0,C 180,E1 -8491.525,E2 -8491.525} C_VEL
LIN {X 0,Y 453.492,Z 459.996,A -85,B 0,C 180,E1 -8494.778,E2 -8494.778} C_VEL
LIN {X 0,Y 453.474,Z 459.999,A -85,B 0,C 180,E1 -8498.311,E2 -8498.311} C_VEL
LIN {X 0,Y 453.497,Z 459.996,A -85,B 0,C 180,E1 -8500.609,E2 -8500.609} C_VEL
LIN {X 0,Y 453.466,Z 459.999,A -85,B 0,C 180,E1 -8503.245,E2 -8503.245} C_VEL
LIN {X 0,Y 453.469,Z 459.999,A -85,B 0,C 180,E1 -8505.779,E2 -8505.779} C_VEL
LIN {X 0,Y 453.482,Z 460,A -85,B 0,C 180,E1 -8508.21,E2 -8508.21} C_VEL
LIN {X 0,Y 453.513,Z 459.995,A -85,B 0,C 180,E1 -8510.791,E2 -8510.791} C_VEL
LIN {X 0,Y 453.46,Z 460,A -85,B 0,C 180,E1 -8513.918,E2 -8513.918} C_VEL
LIN {X 0,Y 453.486,Z 459.997,A -85,B 0,C 180,E1 -8517.151,E2 -8517.151} C_VEL
LIN {X 0,Y 453.479,Z 460,A -85,B 0,C 180,E1 -8520.269,E2 -8520.269} C_VEL
LIN {X 0,Y 453.51,Z 459.993,A -85,B 0,C 180,E1 -8523.294,E2 -8523.294} C_VEL
LIN {X 0,Y 453.507,Z 459.995,A -85,B 0,C 180,E1 -8526.239,E2 -8526.239} C_VEL
LIN {X 0,Y 453.487,Z 459.994,A -85,B 0,C 180,E1 -8529.118,E2 -8529.118} C_VEL
LIN {X 0,Y 453.508,Z 459.996,A -85,B 0,C 180,E1 -8531.944,E2 -8531.944} C_VEL
LIN {X 0,Y 453.544,Z 459.99,A -85,B 0,C 180,E1 -8534.727,E2 -8534.727} C_VEL
LIN {X 0,Y 453.564,Z 459.987,A -85,B 0,C 180,E1 -8538.379,E2 -8538.379} C_VEL
LIN {X 0,Y 453.596,Z 459.983,A -85,B 0,C 180,E1 -8541.087,E2 -8541.087} C_VEL
LIN {X 0,Y 453.599,Z 459.981,A -85,B 0,C 180,E1 -8543.087,E2 -8543.087} C_VEL
LIN {X 0,Y 452.929,Z 460.068,A -85,B 0,C 180,E1 -8543.828,E2 -8543.828} C_VEL
LIN {X 0,Y 449.998,Z 460.43,A -85,B 0,C 180,E1 -8545.03,E2 -8545.03} C_VEL
LIN {X 0,Y 447.579,Z 460.734,A -85,B 0,C 180,E1 -8546,E2 -8546} C_VEL
LIN {X 0,Y 446.637,Z 460.851,A -85,B 0,C 180,E1 -8546.751,E2 -8546.751} C_VEL
LIN {X 0,Y 446.614,Z 460.852,A -85,B 0,C 180,E1 -8547.004,E2 -8547.004} C_VEL
LIN {X 0,Y 446.798,Z 460.832,A -85,B 0,C 180,E1 -8550,E2 -8550} C_VEL
LIN {X 0,Y 446.696,Z 460.842,A -85,B 0,C 180,E1 -8552.705,E2 -8552.705} C_VEL
LIN {X 0,Y 446.646,Z 460.851,A -85,B 0,C 180,E1 -8556.324,E2 -8556.324} C_VEL
LIN {X 0,Y 446.539,Z 460.86,A -85,B 0,C 180,E1 -8559.055,E2 -8559.055} C_VEL
LIN {X 0,Y 446.526,Z 460.864,A -85,B 0,C 180,E1 -8562.73,E2 -8562.73} C_VEL
LIN {X 0,Y 446.501,Z 460.867,A -85,B 0,C 180,E1 -8566.228,E2 -8566.228} C_VEL
LIN {X 0,Y 446.474,Z 460.872,A -85,B 0,C 180,E1 -8569.303,E2 -8569.303} C_VEL
LIN {X 0,Y 446.423,Z 460.878,A -85,B 0,C 180,E1 -8572.2,E2 -8572.2} C_VEL
LIN {X 0,Y 446.462,Z 460.872,A -85,B 0,C 180,E1 -8575.152,E2 -8575.152} C_VEL
LIN {X 0,Y 446.489,Z 460.871,A -85,B 0,C 180,E1 -8578.179,E2 -8578.179} C_VEL
LIN {X 0,Y 446.424,Z 460.878,A -85,B 0,C 180,E1 -8581.775,E2 -8581.775} C_VEL
LIN {X 0,Y 446.433,Z 460.876,A -85,B 0,C 180,E1 -8584.523,E2 -8584.523} C_VEL
LIN {X 0,Y 446.434,Z 460.876,A -85,B 0,C 180,E1 -8588.082,E2 -8588.082} C_VEL
LIN {X 0,Y 446.431,Z 460.876,A -85,B 0,C 180,E1 -8590.918,E2 -8590.918} C_VEL
LIN {X 0,Y 446.404,Z 460.883,A -85,B 0,C 180,E1 -8593.846,E2 -8593.846} C_VEL
LIN {X 0,Y 446.402,Z 460.879,A -85,B 0,C 180,E1 -8596.403,E2 -8596.403} C_VEL
LIN {X 0,Y 446.431,Z 460.877,A -85,B 0,C 180,E1 -8599.082,E2 -8599.082} C_VEL
LIN {X 0,Y 446.41,Z 460.878,A -85,B 0,C 180,E1 -8602.121,E2 -8602.121} C_VEL
LIN {X 0,Y 446.323,Z 460.89,A -85,B 0,C 180,E1 -8604.967,E2 -8604.967} C_VEL
LIN {X 0,Y 445.977,Z 460.935,A -85,B 0,C 180,E1 -8608.317,E2 -8608.317} C_VEL
LIN {X 0,Y 445.777,Z 461.088,A -85,B 0,C 180,E1 -8610.126,E2 -8610.126} C_VEL
LIN {X 0,Y 445.719,Z 463.798,A -85,B 0,C 180,E1 -8612.789,E2 -8612.789} C_VEL
LIN {X 0,Y 445.686,Z 465.888,A -85,B 0,C 180,E1 -8614.801,E2 -8614.801} C_VEL
LIN {X 0,Y 445.587,Z 468.994,A -85,B 0,C 180,E1 -8617.756,E2 -8617.756} C_VEL
LIN {X 0,Y 445.581,Z 472.634,A -85,B 0,C 180,E1 -8621.15,E2 -8621.15} C_VEL
LIN {X 0,Y 445.569,Z 475.834,A -85,B 0,C 180,E1 -8624.082,E2 -8624.082} C_VEL
LIN {X 0,Y 448.72,Z 490.01,A -85,B 0,C 180,E1 -8624.674,E2 -8624.674} C_VEL
LIN {X 0,Y 449.392,Z 493.974,A -85,B 0,C 180,E1 -8624.872,E2 -8624.872} C_VEL
LIN {X 0,Y 448.983,Z 505.815,A -85,B 0,C 180,E1 -8625.496,E2 -8625.496} C_VEL
LIN {X 0,Y 448.445,Z 517.963,A -85,B 0,C 180,E1 -8626.328,E2 -8626.328} C_VEL
LIN {X 0,Y 447.929,Z 529.179,A -85,B 0,C 180,E1 -8627.311,E2 -8627.311} C_VEL
LIN {X 0,Y 447.314,Z 539.654,A -85,B 0,C 180,E1 -8628.444,E2 -8628.444} C_VEL
LIN {X 0,Y 446.85,Z 548.16,A -85,B 0,C 180,E1 -8629.579,E2 -8629.579} C_VEL
LIN {X 0,Y 446.424,Z 556.47,A -85,B 0,C 180,E1 -8630.942,E2 -8630.942} C_VEL
LIN {X 0,Y 446.032,Z 563.175,A -85,B 0,C 180,E1 -8632.303,E2 -8632.303} C_VEL
LIN {X 0,Y 445.913,Z 568.52,A -85,B 0,C 180,E1 -8633.666,E2 -8633.666} C_VEL
LIN {X 0,Y 445.624,Z 572.691,A -85,B 0,C 180,E1 -8635.024,E2 -8635.024} C_VEL
LIN {X 0,Y 445.608,Z 575.782,A -85,B 0,C 180,E1 -8636.383,E2 -8636.383} C_VEL
LIN {X 0,Y 445.546,Z 577.304,A -85,B 0,C 180,E1 -8637.287,E2 -8637.287} C_VEL
LIN {X 0,Y 445.502,Z 578.383,A -85,B 0,C 180,E1 -8638.192,E2 -8638.192} C_VEL
LIN {X 0,Y 445.401,Z 579.377,A -85,B 0,C 180,E1 -8640,E2 -8640} C_VEL
LIN {X 0,Y 445.428,Z 579.244,A -85,B 0,C 180,E1 -8640.904,E2 -8640.904} C_VEL
LIN {X 0,Y 445.521,Z 578.695,A -85,B 0,C 180,E1 -8641.808,E2 -8641.808} C_VEL
LIN {X 0,Y 445.572,Z 577.76,A -85,B 0,C 180,E1 -8642.712,E2 -8642.712} C_VEL
LIN {X 0,Y 445.62,Z 576.427,A -85,B 0,C 180,E1 -8643.617,E2 -8643.617} C_VEL
LIN {X 0,Y 445.679,Z 573.584,A -85,B 0,C 180,E1 -8644.975,E2 -8644.975} C_VEL
LIN {X 0,Y 445.94,Z 569.687,A -85,B 0,C 180,E1 -8646.334,E2 -8646.334} C_VEL
LIN {X 0,Y 446.134,Z 564.645,A -85,B 0,C 180,E1 -8647.695,E2 -8647.695} C_VEL
LIN {X 0,Y 446.516,Z 558.256,A -85,B 0,C 180,E1 -8649.056,E2 -8649.056} C_VEL
LIN {X 0,Y 446.975,Z 550.314,A -85,B 0,C 180,E1 -8650.417,E2 -8650.417} C_VEL
LIN {X 0,Y 447.423,Z 542.246,A -85,B 0,C 180,E1 -8651.553,E2 -8651.553} C_VEL
LIN {X 0,Y 448.09,Z 532.404,A -85,B 0,C 180,E1 -8652.684,E2 -8652.684} C_VEL
LIN {X 0,Y 448.613,Z 521.516,A -85,B 0,C 180,E1 -8653.695,E2 -8653.695} C_VEL
LIN {X 0,Y 449.169,Z 510.737,A -85,B 0,C 180,E1 -8654.498,E2 -8654.498} C_VEL
LIN {X 0,Y 449.726,Z 498.058,A -85,B 0,C 180,E1 -8655.232,E2 -8655.232} C_VEL
LIN {X 0,Y 449.687,Z 493.545,A -85,B 0,C 180,E1 -8655.456,E2 -8655.456} C_VEL
LIN {X 0,Y 446.822,Z 481.985,A -85,B 0,C 180,E1 -8656.04,E2 -8656.04} C_VEL
LIN {X 0,Y 445.842,Z 478.438,A -85,B 0,C 180,E1 -8656.213,E2 -8656.213} C_VEL
LIN {X 0,Y 445.903,Z 475.667,A -85,B 0,C 180,E1 -8659.329,E2 -8659.329} C_VEL
LIN {X 0,Y 445.999,Z 473.255,A -85,B 0,C 180,E1 -8662.222,E2 -8662.222} C_VEL
LIN {X 0,Y 446.17,Z 470.936,A -85,B 0,C 180,E1 -8665.17,E2 -8665.17} C_VEL
LIN {X 0,Y 446.408,Z 468.762,A -85,B 0,C 180,E1 -8668.184,E2 -8668.184} C_VEL
LIN {X 0,Y 446.668,Z 466.49,A -85,B 0,C 180,E1 -8671.826,E2 -8671.826} C_VEL
LIN {X 0,Y 446.822,Z 465.157,A -85,B 0,C 180,E1 -8674.488,E2 -8674.488} C_VEL
LIN {X 0,Y 446.897,Z 464.342,A -85,B 0,C 180,E1 -8676.698,E2 -8676.698} C_VEL
LIN {X 0,Y 446.896,Z 463.795,A -85,B 0,C 180,E1 -8679.593,E2 -8679.593} C_VEL
LIN {X 0,Y 446.984,Z 463.977,A -85,B 0,C 180,E1 -8682.539,E2 -8682.539} C_VEL
LIN {X 0,Y 447.13,Z 464.804,A -85,B 0,C 180,E1 -8685.017,E2 -8685.017} C_VEL
LIN {X 0,Y 447.44,Z 466.492,A -85,B 0,C 180,E1 -8687.581,E2 -8687.581} C_VEL
LIN {X 0,Y 447.909,Z 469.086,A -85,B 0,C 180,E1 -8690.25,E2 -8690.25} C_VEL
LIN {X 0,Y 448.298,Z 471.711,A -85,B 0,C 180,E1 -8692.308,E2 -8692.308} C_VEL
LIN {X 0,Y 448.404,Z 475.217,A -85,B 0,C 180,E1 -8694.555,E2 -8694.555} C_VEL
LIN {X 0,Y 448.004,Z 479.175,A -85,B 0,C 180,E1 -8696.697,E2 -8696.697} C_VEL
LIN {X 0,Y 447.317,Z 485.704,A -85,B 0,C 180,E1 -8699.817,E2 -8699.817} C_VEL
LIN {X 0,Y 446.841,Z 492.778,A -85,B 0,C 180,E1 -8702.863,E2 -8702.863} C_VEL
LIN {X 0,Y 446.421,Z 500.465,A -85,B 0,C 180,E1 -8705.937,E2 -8705.937} C_VEL
LIN {X 0,Y 446.115,Z 509.22,A -85,B 0,C 180,E1 -8709.239,E2 -8709.239} C_VEL
LIN {X 0,Y 445.858,Z 518.391,A -85,B 0,C 180,E1 -8712.573,E2 -8712.573} C_VEL
LIN {X 0,Y 445.799,Z 521.662,A -85,B 0,C 180,E1 -8713.734,E2 -8713.734} C_VEL
LIN {X 0,Y 447.725,Z 535.029,A -85,B 0,C 180,E1 -8714.246,E2 -8714.246} C_VEL
LIN {X 0,Y 448.991,Z 548.698,A -85,B 0,C 180,E1 -8714.916,E2 -8714.916} C_VEL
LIN {X 0,Y 448.342,Z 561.955,A -85,B 0,C 180,E1 -8715.706,E2 -8715.706} C_VEL
LIN {X 0,Y 447.771,Z 572.802,A -85,B 0,C 180,E1 -8716.534,E2 -8716.534} C_VEL
LIN {X 0,Y 447.107,Z 584.352,A -85,B 0,C 180,E1 -8717.633,E2 -8717.633} C_VEL
LIN {X 0,Y 446.677,Z 593.17,A -85,B 0,C 180,E1 -8718.657,E2 -8718.657} C_VEL
LIN {X 0,Y 446.212,Z 601.34,A -85,B 0,C 180,E1 -8719.794,E2 -8719.794} C_VEL
LIN {X 0,Y 445.881,Z 609.385,A -85,B 0,C 180,E1 -8721.16,E2 -8721.16} C_VEL
LIN {X 0,Y 445.694,Z 614.889,A -85,B 0,C 180,E1 -8722.297,E2 -8722.297} C_VEL
LIN {X 0,Y 445.494,Z 621.134,A -85,B 0,C 180,E1 -8723.927,E2 -8723.927} C_VEL
LIN {X 0,Y 445.432,Z 625.557,A -85,B 0,C 180,E1 -8725.475,E2 -8725.475} C_VEL
LIN {X 0,Y 445.441,Z 627.53,A -85,B 0,C 180,E1 -8726.382,E2 -8726.382} C_VEL
LIN {X 0,Y 445.475,Z 629.017,A -85,B 0,C 180,E1 -8727.287,E2 -8727.287} C_VEL
LIN {X 0,Y 445.452,Z 630.085,A -85,B 0,C 180,E1 -8728.192,E2 -8728.192} C_VEL
LIN {X 0,Y 445.427,Z 630.749,A -85,B 0,C 180,E1 -8729.096,E2 -8729.096} C_VEL
LIN {X 0,Y 445.399,Z 630.995,A -85,B 0,C 180,E1 -8730,E2 -8730} C_VEL
LIN {X 0,Y 445.427,Z 630.793,A -85,B 0,C 180,E1 -8730.904,E2 -8730.904} C_VEL
LIN {X 0,Y 445.45,Z 630.19,A -85,B 0,C 180,E1 -8731.808,E2 -8731.808} C_VEL
LIN {X 0,Y 445.467,Z 629.185,A -85,B 0,C 180,E1 -8732.713,E2 -8732.713} C_VEL
LIN {X 0,Y 445.428,Z 627.735,A -85,B 0,C 180,E1 -8733.618,E2 -8733.618} C_VEL
LIN {X 0,Y 445.492,Z 624.724,A -85,B 0,C 180,E1 -8734.978,E2 -8734.978} C_VEL
LIN {X 0,Y 445.529,Z 620.461,A -85,B 0,C 180,E1 -8736.385,E2 -8736.385} C_VEL
LIN {X 0,Y 445.721,Z 614.317,A -85,B 0,C 180,E1 -8737.93,E2 -8737.93} C_VEL
LIN {X 0,Y 446.029,Z 607.446,A -85,B 0,C 180,E1 -8739.294,E2 -8739.294} C_VEL
LIN {X 0,Y 446.402,Z 598.879,A -85,B 0,C 180,E1 -8740.66,E2 -8740.66} C_VEL
LIN {X 0,Y 446.942,Z 590.101,A -85,B 0,C 180,E1 -8741.795,E2 -8741.795} C_VEL
LIN {X 0,Y 447.481,Z 579.86,A -85,B 0,C 180,E1 -8742.882,E2 -8742.882} C_VEL
LIN {X 0,Y 448.063,Z 568.664,A -85,B 0,C 180,E1 -8743.839,E2 -8743.839} C_VEL
LIN {X 0,Y 448.628,Z 556.85,A -85,B 0,C 180,E1 -8744.632,E2 -8744.632} C_VEL
LIN {X 0,Y 449.008,Z 547.279,A -85,B 0,C 180,E1 -8745.141,E2 -8745.141} C_VEL
LIN {X 0,Y 447.276,Z 533.473,A -85,B 0,C 180,E1 -8745.753,E2 -8745.753} C_VEL
LIN {X 0,Y 445.869,Z 523.917,A -85,B 0,C 180,E1 -8746.068,E2 -8746.068} C_VEL
LIN {X 0,Y 446.1,Z 515.023,A -85,B 0,C 180,E1 -8749.32,E2 -8749.32} C_VEL
LIN {X 0,Y 446.426,Z 505.99,A -85,B 0,C 180,E1 -8752.687,E2 -8752.687} C_VEL
LIN {X 0,Y 446.889,Z 496.952,A -85,B 0,C 180,E1 -8756.126,E2 -8756.126} C_VEL
LIN {X 0,Y 447.329,Z 489.221,A -85,B 0,C 180,E1 -8759.146,E2 -8759.146} C_VEL
LIN {X 0,Y 447.858,Z 481.494,A -85,B 0,C 180,E1 -8762.245,E2 -8762.245} C_VEL
LIN {X 0,Y 448.317,Z 473.926,A -85,B 0,C 180,E1 -8765.395,E2 -8765.395} C_VEL
LIN {X 0,Y 448.155,Z 470.498,A -85,B 0,C 180,E1 -8766.89,E2 -8766.89} C_VEL
LIN {X 0,Y 446.94,Z 463.436,A -85,B 0,C 180,E1 -8770.144,E2 -8770.144} C_VEL
LIN {X 0,Y 446.446,Z 460.877,A -85,B 0,C 180,E1 -8771.389,E2 -8771.389} C_VEL
LIN {X 0,Y 446.458,Z 460.873,A -85,B 0,C 180,E1 -8775.103,E2 -8775.103} C_VEL
LIN {X 0,Y 446.438,Z 460.875,A -85,B 0,C 180,E1 -8778.61,E2 -8778.61} C_VEL
LIN {X 0,Y 446.443,Z 460.875,A -85,B 0,C 180,E1 -8780.973,E2 -8780.973} C_VEL
LIN {X 0,Y 446.42,Z 460.878,A -85,B 0,C 180,E1 -8784.374,E2 -8784.374} C_VEL
LIN {X 0,Y 446.423,Z 460.875,A -85,B 0,C 180,E1 -8787.639,E2 -8787.639} C_VEL
LIN {X 0,Y 446.451,Z 460.874,A -85,B 0,C 180,E1 -8790.791,E2 -8790.791} C_VEL
LIN {X 0,Y 446.479,Z 460.869,A -85,B 0,C 180,E1 -8793.849,E2 -8793.849} C_VEL
LIN {X 0,Y 446.43,Z 460.876,A -85,B 0,C 180,E1 -8796.823,E2 -8796.823} C_VEL
LIN {X 0,Y 446.447,Z 460.874,A -85,B 0,C 180,E1 -8799.737,E2 -8799.737} C_VEL
LIN {X 0,Y 446.466,Z 460.875,A -85,B 0,C 180,E1 -8802.597,E2 -8802.597} C_VEL
LIN {X 0,Y 446.472,Z 460.871,A -85,B 0,C 180,E1 -8805.413,E2 -8805.413} C_VEL
LIN {X 0,Y 446.519,Z 460.865,A -85,B 0,C 180,E1 -8808.193,E2 -8808.193} C_VEL
LIN {X 0,Y 446.602,Z 460.854,A -85,B 0,C 180,E1 -8811.858,E2 -8811.858} C_VEL
LIN {X 0,Y 446.647,Z 460.85,A -85,B 0,C 180,E1 -8814.583,E2 -8814.583} C_VEL
LIN {X 0,Y 446.666,Z 460.848,A -85,B 0,C 180,E1 -8818.197,E2 -8818.197} C_VEL
LIN {X 0,Y 446.797,Z 460.832,A -85,B 0,C 180,E1 -8820,E2 -8820} C_VEL
LIN {X 0,Y 446.71,Z 460.844,A -85,B 0,C 180,E1 -8822.705,E2 -8822.705} C_VEL
LIN {X 0,Y 446.649,Z 460.851,A -85,B 0,C 180,E1 -8826.324,E2 -8826.324} C_VEL
LIN {X 0,Y 446.541,Z 460.863,A -85,B 0,C 180,E1 -8829.056,E2 -8829.056} C_VEL
LIN {X 0,Y 446.524,Z 460.864,A -85,B 0,C 180,E1 -8832.73,E2 -8832.73} C_VEL
LIN {X 0,Y 446.499,Z 460.868,A -85,B 0,C 180,E1 -8836.228,E2 -8836.228} C_VEL
LIN {X 0,Y 446.472,Z 460.869,A -85,B 0,C 180,E1 -8839.303,E2 -8839.303} C_VEL
LIN {X 0,Y 446.421,Z 460.878,A -85,B 0,C 180,E1 -8842.2,E2 -8842.2} C_VEL
LIN {X 0,Y 446.46,Z 460.871,A -85,B 0,C 180,E1 -8845.152,E2 -8845.152} C_VEL
LIN {X 0,Y 446.487,Z 460.871,A -85,B 0,C 180,E1 -8848.179,E2 -8848.179} C_VEL
LIN {X 0,Y 446.422,Z 460.876,A -85,B 0,C 180,E1 -8851.775,E2 -8851.775} C_VEL
LIN {X 0,Y 446.433,Z 460.876,A -85,B 0,C 180,E1 -8854.523,E2 -8854.523} C_VEL
LIN {X 0,Y 446.432,Z 460.876,A -85,B 0,C 180,E1 -8858.082,E2 -8858.082} C_VEL
LIN {X 0,Y 446.43,Z 460.874,A -85,B 0,C 180,E1 -8860.918,E2 -8860.918} C_VEL
LIN {X 0,Y 446.426,Z 460.878,A -85,B 0,C 180,E1 -8863.843,E2 -8863.843} C_VEL
LIN {X 0,Y 446.418,Z 460.88,A -85,B 0,C 180,E1 -8866.401,E2 -8866.401} C_VEL
LIN {X 0,Y 446.451,Z 460.875,A -85,B 0,C 180,E1 -8869.803,E2 -8869.803} C_VEL
LIN {X 0,Y 446.431,Z 460.876,A -85,B 0,C 180,E1 -8872.123,E2 -8872.123} C_VEL
LIN {X 0,Y 446.434,Z 460.874,A -85,B 0,C 180,E1 -8875.477,E2 -8875.477} C_VEL
LIN {X 0,Y 446.42,Z 460.879,A -85,B 0,C 180,E1 -8878.7,E2 -8878.7} C_VEL
LIN {X 0,Y 446.488,Z 460.869,A -85,B 0,C 180,E1 -8881.822,E2 -8881.822} C_VEL
LIN {X 0,Y 446.462,Z 460.873,A -85,B 0,C 180,E1 -8884.848,E2 -8884.848} C_VEL
LIN {X 0,Y 446.452,Z 460.876,A -85,B 0,C 180,E1 -8888.245,E2 -8888.245} C_VEL
LIN {X 0,Y 446.457,Z 460.874,A -85,B 0,C 180,E1 -8891.649,E2 -8891.649} C_VEL
LIN {X 0,Y 446.512,Z 460.868,A -85,B 0,C 180,E1 -8894.48,E2 -8894.48} C_VEL
LIN {X 0,Y 446.522,Z 460.865,A -85,B 0,C 180,E1 -8898.193,E2 -8898.193} C_VEL
LIN {X 0,Y 446.542,Z 460.862,A -85,B 0,C 180,E1 -8900.945,E2 -8900.945} C_VEL
LIN {X 0,Y 446.624,Z 460.852,A -85,B 0,C 180,E1 -8903.676,E2 -8903.676} C_VEL
LIN {X 0,Y 446.614,Z 460.852,A -85,B 0,C 180,E1 -8907.004,E2 -8907.004} C_VEL
LIN {X 0,Y 446.088,Z 460.92,A -85,B 0,C 180,E1 -8907.757,E2 -8907.757} C_VEL
LIN {X 0,Y 443.267,Z 461.271,A -85,B 0,C 180,E1 -8908.98,E2 -8908.98} C_VEL
LIN {X 0,Y 440.786,Z 461.581,A -85,B 0,C 180,E1 -8909.967,E2 -8909.967} C_VEL
LIN {X 0,Y 439.705,Z 461.712,A -85,B 0,C 180,E1 -8910.731,E2 -8910.731} C_VEL
LIN {X 0,Y 439.614,Z 461.722,A -85,B 0,C 180,E1 -8910.99,E2 -8910.99} C_VEL
LIN {X 0,Y 439.645,Z 461.721,A -85,B 0,C 180,E1 -8912.749,E2 -8912.749} C_VEL
LIN {X 0,Y 439.618,Z 461.726,A -85,B 0,C 180,E1 -8916.425,E2 -8916.425} C_VEL
LIN {X 0,Y 439.502,Z 461.737,A -85,B 0,C 180,E1 -8919.202,E2 -8919.202} C_VEL
LIN {X 0,Y 439.47,Z 461.742,A -85,B 0,C 180,E1 -8922.938,E2 -8922.938} C_VEL
LIN {X 0,Y 439.452,Z 461.745,A -85,B 0,C 180,E1 -8926.349,E2 -8926.349} C_VEL
LIN {X 0,Y 439.407,Z 461.751,A -85,B 0,C 180,E1 -8929.626,E2 -8929.626} C_VEL
LIN {X 0,Y 439.37,Z 461.753,A -85,B 0,C 180,E1 -8932.575,E2 -8932.575} C_VEL
LIN {X 0,Y 439.41,Z 461.752,A -85,B 0,C 180,E1 -8935.585,E2 -8935.585} C_VEL
LIN {X 0,Y 439.422,Z 461.748,A -85,B 0,C 180,E1 -8938.673,E2 -8938.673} C_VEL
LIN {X 0,Y 439.375,Z 461.755,A -85,B 0,C 180,E1 -8942.03,E2 -8942.03} C_VEL
LIN {X 0,Y 439.399,Z 461.752,A -85,B 0,C 180,E1 -8945.34,E2 -8945.34} C_VEL
LIN {X 0,Y 439.393,Z 461.752,A -85,B 0,C 180,E1 -8948.594,E2 -8948.594} C_VEL
LIN {X 0,Y 439.392,Z 461.754,A -85,B 0,C 180,E1 -8951.257,E2 -8951.257} C_VEL
LIN {X 0,Y 439.404,Z 461.749,A -85,B 0,C 180,E1 -8954.729,E2 -8954.729} C_VEL
LIN {X 0,Y 439.4,Z 461.752,A -85,B 0,C 180,E1 -8957.796,E2 -8957.796} C_VEL
LIN {X 0,Y 439.43,Z 461.748,A -85,B 0,C 180,E1 -8960.227,E2 -8960.227} C_VEL
LIN {X 0,Y 439.345,Z 461.76,A -85,B 0,C 180,E1 -8963.71,E2 -8963.71} C_VEL
LIN {X 0,Y 439.12,Z 461.788,A -85,B 0,C 180,E1 -8966.331,E2 -8966.331} C_VEL
LIN {X 0,Y 438.801,Z 461.829,A -85,B 0,C 180,E1 -8969.168,E2 -8969.168} C_VEL
LIN {X 0,Y 438.706,Z 461.858,A -85,B 0,C 180,E1 -8970.223,E2 -8970.223} C_VEL
LIN {X 0,Y 438.651,Z 465.035,A -85,B 0,C 180,E1 -8973.345,E2 -8973.345} C_VEL
LIN {X 0,Y 438.587,Z 468.184,A -85,B 0,C 180,E1 -8976.384,E2 -8976.384} C_VEL
LIN {X 0,Y 438.512,Z 471.319,A -85,B 0,C 180,E1 -8979.354,E2 -8979.354} C_VEL
LIN {X 0,Y 438.467,Z 474.448,A -85,B 0,C 180,E1 -8982.269,E2 -8982.269} C_VEL
LIN {X 0,Y 438.475,Z 476.172,A -85,B 0,C 180,E1 -8983.846,E2 -8983.846} C_VEL
LIN {X 0,Y 441.786,Z 490.947,A -85,B 0,C 180,E1 -8984.487,E2 -8984.487} C_VEL
LIN {X 0,Y 442.475,Z 494.836,A -85,B 0,C 180,E1 -8984.689,E2 -8984.689} C_VEL
LIN {X 0,Y 441.994,Z 507.484,A -85,B 0,C 180,E1 -8985.379,E2 -8985.379} C_VEL
LIN {X 0,Y 441.42,Z 519.841,A -85,B 0,C 180,E1 -8986.271,E2 -8986.271} C_VEL
LIN {X 0,Y 440.83,Z 531.487,A -85,B 0,C 180,E1 -8987.337,E2 -8987.337} C_VEL
LIN {X 0,Y 440.236,Z 541.531,A -85,B 0,C 180,E1 -8988.489,E2 -8988.489} C_VEL
LIN {X 0,Y 439.682,Z 551.284,A -85,B 0,C 180,E1 -8989.873,E2 -8989.873} C_VEL
LIN {X 0,Y 439.242,Z 559.077,A -85,B 0,C 180,E1 -8991.257,E2 -8991.257} C_VEL
LIN {X 0,Y 438.919,Z 565.332,A -85,B 0,C 180,E1 -8992.64,E2 -8992.64} C_VEL
LIN {X 0,Y 438.766,Z 570.301,A -85,B 0,C 180,E1 -8994.024,E2 -8994.024} C_VEL
LIN {X 0,Y 438.567,Z 574.139,A -85,B 0,C 180,E1 -8995.404,E2 -8995.404} C_VEL
LIN {X 0,Y 438.55,Z 576.126,A -85,B 0,C 180,E1 -8996.325,E2 -8996.325} C_VEL
LIN {X 0,Y 438.473,Z 577.677,A -85,B 0,C 180,E1 -8997.244,E2 -8997.244} C_VEL
LIN {X 0,Y 438.368,Z 579.477,A -85,B 0,C 180,E1 -8999.081,E2 -8999.081} C_VEL
LIN {X 0,Y 438.339,Z 579.793,A -85,B 0,C 180,E1 -9000,E2 -9000} C_VEL
LIN {X 0,Y 438.368,Z 579.68,A -85,B 0,C 180,E1 -9000.918,E2 -9000.918} C_VEL
LIN {X 0,Y 438.465,Z 579.141,A -85,B 0,C 180,E1 -9001.837,E2 -9001.837} C_VEL
LIN {X 0,Y 438.497,Z 578.217,A -85,B 0,C 180,E1 -9002.756,E2 -9002.756} C_VEL
LIN {X 0,Y 438.567,Z 576.892,A -85,B 0,C 180,E1 -9003.675,E2 -9003.675} C_VEL
LIN {X 0,Y 438.623,Z 574.061,A -85,B 0,C 180,E1 -9005.056,E2 -9005.056} C_VEL
LIN {X 0,Y 438.901,Z 570.182,A -85,B 0,C 180,E1 -9006.436,E2 -9006.436} C_VEL
LIN {X 0,Y 439.109,Z 565.178,A -85,B 0,C 180,E1 -9007.819,E2 -9007.819} C_VEL
LIN {X 0,Y 439.541,Z 558.838,A -85,B 0,C 180,E1 -9009.201,E2 -9009.201} C_VEL
LIN {X 0,Y 440.029,Z 550.946,A -85,B 0,C 180,E1 -9010.584,E2 -9010.584} C_VEL
LIN {X 0,Y 440.497,Z 542.909,A -85,B 0,C 180,E1 -9011.737,E2 -9011.737} C_VEL
LIN {X 0,Y 441.202,Z 533.121,A -85,B 0,C 180,E1 -9012.886,E2 -9012.886} C_VEL
LIN {X 0,Y 441.818,Z 521.35,A -85,B 0,C 180,E1 -9013.991,E2 -9013.991} C_VEL
LIN {X 0,Y 442.441,Z 509.992,A -85,B 0,C 180,E1 -9014.841,E2 -9014.841} C_VEL
LIN {X 0,Y 443.025,Z 496.976,A -85,B 0,C 180,E1 -9015.586,E2 -9015.586} C_VEL
LIN {X 0,Y 442.622,Z 493.059,A -85,B 0,C 180,E1 -9015.798,E2 -9015.798} C_VEL
LIN {X 0,Y 439.419,Z 481.316,A -85,B 0,C 180,E1 -9016.417,E2 -9016.417} C_VEL
LIN {X 0,Y 438.787,Z 479.026,A -85,B 0,C 180,E1 -9016.528,E2 -9016.528} C_VEL
LIN {X 0,Y 438.857,Z 476.321,A -85,B 0,C 180,E1 -9019.652,E2 -9019.652} C_VEL
LIN {X 0,Y 438.986,Z 473.936,A -85,B 0,C 180,E1 -9022.596,E2 -9022.596} C_VEL
LIN {X 0,Y 439.168,Z 471.672,A -85,B 0,C 180,E1 -9025.6,E2 -9025.6} C_VEL
LIN {X 0,Y 439.39,Z 469.559,A -85,B 0,C 180,E1 -9028.675,E2 -9028.675} C_VEL
LIN {X 0,Y 439.698,Z 467.553,A -85,B 0,C 180,E1 -9032.098,E2 -9032.098} C_VEL
LIN {X 0,Y 439.899,Z 466.198,A -85,B 0,C 180,E1 -9035.11,E2 -9035.11} C_VEL
LIN {X 0,Y 439.939,Z 465.534,A -85,B 0,C 180,E1 -9037.376,E2 -9037.376} C_VEL
LIN {X 0,Y 439.967,Z 465.224,A -85,B 0,C 180,E1 -9039.937,E2 -9039.937} C_VEL
LIN {X 0,Y 440.052,Z 465.552,A -85,B 0,C 180,E1 -9042.721,E2 -9042.721} C_VEL
LIN {X 0,Y 440.232,Z 466.576,A -85,B 0,C 180,E1 -9045.377,E2 -9045.377} C_VEL
LIN {X 0,Y 440.583,Z 468.355,A -85,B 0,C 180,E1 -9047.935,E2 -9047.935} C_VEL
LIN {X 0,Y 441.003,Z 470.783,A -85,B 0,C 180,E1 -9050.397,E2 -9050.397} C_VEL
LIN {X 0,Y 441.439,Z 473.841,A -85,B 0,C 180,E1 -9052.772,E2 -9052.772} C_VEL
LIN {X 0,Y 441.346,Z 477.425,A -85,B 0,C 180,E1 -9055.022,E2 -9055.022} C_VEL
LIN {X 0,Y 440.875,Z 481.441,A -85,B 0,C 180,E1 -9057.18,E2 -9057.18} C_VEL
LIN {X 0,Y 440.372,Z 486.241,A -85,B 0,C 180,E1 -9059.519,E2 -9059.519} C_VEL
LIN {X 0,Y 439.801,Z 493.901,A -85,B 0,C 180,E1 -9062.907,E2 -9062.907} C_VEL
LIN {X 0,Y 439.382,Z 500.813,A -85,B 0,C 180,E1 -9065.745,E2 -9065.745} C_VEL
LIN {X 0,Y 439.097,Z 508.906,A -85,B 0,C 180,E1 -9068.892,E2 -9068.892} C_VEL
LIN {X 0,Y 438.775,Z 518.035,A -85,B 0,C 180,E1 -9072.282,E2 -9072.282} C_VEL
LIN {X 0,Y 438.762,Z 521.163,A -85,B 0,C 180,E1 -9073.421,E2 -9073.421} C_VEL
LIN {X 0,Y 440.794,Z 535.009,A -85,B 0,C 180,E1 -9073.968,E2 -9073.968} C_VEL
LIN {X 0,Y 442.138,Z 548.79,A -85,B 0,C 180,E1 -9074.677,E2 -9074.677} C_VEL
LIN {X 0,Y 441.453,Z 561.849,A -85,B 0,C 180,E1 -9075.478,E2 -9075.478} C_VEL
LIN {X 0,Y 440.82,Z 572.827,A -85,B 0,C 180,E1 -9076.342,E2 -9076.342} C_VEL
LIN {X 0,Y 440.169,Z 584.051,A -85,B 0,C 180,E1 -9077.435,E2 -9077.435} C_VEL
LIN {X 0,Y 439.593,Z 594.587,A -85,B 0,C 180,E1 -9078.706,E2 -9078.706} C_VEL
LIN {X 0,Y 439.065,Z 603.814,A -85,B 0,C 180,E1 -9080.092,E2 -9080.092} C_VEL
LIN {X 0,Y 438.773,Z 611.312,A -85,B 0,C 180,E1 -9081.48,E2 -9081.48} C_VEL
LIN {X 0,Y 438.539,Z 616.392,A -85,B 0,C 180,E1 -9082.634,E2 -9082.634} C_VEL
LIN {X 0,Y 438.393,Z 621.178,A -85,B 0,C 180,E1 -9083.967,E2 -9083.967} C_VEL
LIN {X 0,Y 438.36,Z 625.151,A -85,B 0,C 180,E1 -9085.402,E2 -9085.402} C_VEL
LIN {X 0,Y 438.342,Z 627.12,A -85,B 0,C 180,E1 -9086.323,E2 -9086.323} C_VEL
LIN {X 0,Y 438.4,Z 628.607,A -85,B 0,C 180,E1 -9087.243,E2 -9087.243} C_VEL
LIN {X 0,Y 438.368,Z 629.675,A -85,B 0,C 180,E1 -9088.162,E2 -9088.162} C_VEL
LIN {X 0,Y 438.366,Z 630.34,A -85,B 0,C 180,E1 -9089.081,E2 -9089.081} C_VEL
LIN {X 0,Y 438.337,Z 630.577,A -85,B 0,C 180,E1 -9090,E2 -9090} C_VEL
LIN {X 0,Y 438.366,Z 630.371,A -85,B 0,C 180,E1 -9090.919,E2 -9090.919} C_VEL
LIN {X 0,Y 438.366,Z 629.762,A -85,B 0,C 180,E1 -9091.837,E2 -9091.837} C_VEL
LIN {X 0,Y 438.392,Z 628.752,A -85,B 0,C 180,E1 -9092.757,E2 -9092.757} C_VEL
LIN {X 0,Y 438.332,Z 627.284,A -85,B 0,C 180,E1 -9093.677,E2 -9093.677} C_VEL
LIN {X 0,Y 438.422,Z 624.257,A -85,B 0,C 180,E1 -9095.058,E2 -9095.058} C_VEL
LIN {X 0,Y 438.448,Z 620.133,A -85,B 0,C 180,E1 -9096.442,E2 -9096.442} C_VEL
LIN {X 0,Y 438.67,Z 613.798,A -85,B 0,C 180,E1 -9098.058,E2 -9098.058} C_VEL
LIN {X 0,Y 438.967,Z 606.893,A -85,B 0,C 180,E1 -9099.445,E2 -9099.445} C_VEL
LIN {X 0,Y 439.39,Z 598.271,A -85,B 0,C 180,E1 -9100.833,E2 -9100.833} C_VEL
LIN {X 0,Y 439.931,Z 589.447,A -85,B 0,C 180,E1 -9101.986,E2 -9101.986} C_VEL
LIN {X 0,Y 440.488,Z 579.647,A -85,B 0,C 180,E1 -9103.041,E2 -9103.041} C_VEL
LIN {X 0,Y 441.122,Z 567.861,A -85,B 0,C 180,E1 -9104.062,E2 -9104.062} C_VEL
LIN {X 0,Y 441.719,Z 555.968,A -85,B 0,C 180,E1 -9104.866,E2 -9104.866} C_VEL
LIN {X 0,Y 442.014,Z 547.505,A -85,B 0,C 180,E1 -9105.327,E2 -9105.327} C_VEL
LIN {X 0,Y 440.26,Z 533.631,A -85,B 0,C 180,E1 -9105.962,E2 -9105.962} C_VEL
LIN {X 0,Y 438.801,Z 523.575,A -85,B 0,C 180,E1 -9106.322,E2 -9106.322} C_VEL
LIN {X 0,Y 439.043,Z 514.674,A -85,B 0,C 180,E1 -9109.643,E2 -9109.643} C_VEL
LIN {X 0,Y 439.408,Z 505.647,A -85,B 0,C 180,E1 -9113.07,E2 -9113.07} C_VEL
LIN {X 0,Y 439.902,Z 496.653,A -85,B 0,C 180,E1 -9116.573,E2 -9116.573} C_VEL
LIN {X 0,Y 440.369,Z 488.931,A -85,B 0,C 180,E1 -9119.653,E2 -9119.653} C_VEL
LIN {X 0,Y 440.886,Z 481.222,A -85,B 0,C 180,E1 -9122.819,E2 -9122.819} C_VEL
LIN {X 0,Y 441.354,Z 474.436,A -85,B 0,C 180,E1 -9125.697,E2 -9125.697} C_VEL
LIN {X 0,Y 440.817,Z 469.631,A -85,B 0,C 180,E1 -9127.866,E2 -9127.866} C_VEL
LIN {X 0,Y 439.658,Z 463.15,A -85,B 0,C 180,E1 -9130.949,E2 -9130.949} C_VEL
LIN {X 0,Y 439.406,Z 461.753,A -85,B 0,C 180,E1 -9131.7,E2 -9131.7} C_VEL
LIN {X 0,Y 439.41,Z 461.75,A -85,B 0,C 180,E1 -9135.272,E2 -9135.272} C_VEL
LIN {X 0,Y 439.396,Z 461.753,A -85,B 0,C 180,E1 -9138.742,E2 -9138.742} C_VEL
LIN {X 0,Y 439.374,Z 461.753,A -85,B 0,C 180,E1 -9141.608,E2 -9141.608} C_VEL
LIN {X 0,Y 439.4,Z 461.752,A -85,B 0,C 180,E1 -9144.844,E2 -9144.844} C_VEL
LIN {X 0,Y 439.374,Z 461.754,A -85,B 0,C 180,E1 -9148.14,E2 -9148.14} C_VEL
LIN {X 0,Y 439.434,Z 461.747,A -85,B 0,C 180,E1 -9151.598,E2 -9151.598} C_VEL
LIN {X 0,Y 439.406,Z 461.751,A -85,B 0,C 180,E1 -9154.415,E2 -9154.415} C_VEL
LIN {X 0,Y 439.366,Z 461.756,A -85,B 0,C 180,E1 -9157.425,E2 -9157.425} C_VEL
LIN {X 0,Y 439.443,Z 461.748,A -85,B 0,C 180,E1 -9160.663,E2 -9160.663} C_VEL
LIN {X 0,Y 439.464,Z 461.745,A -85,B 0,C 180,E1 -9164.225,E2 -9164.225} C_VEL
LIN {X 0,Y 439.485,Z 461.741,A -85,B 0,C 180,E1 -9168.001,E2 -9168.001} C_VEL
LIN {X 0,Y 439.55,Z 461.732,A -85,B 0,C 180,E1 -9171.726,E2 -9171.726} C_VEL
LIN {X 0,Y 439.623,Z 461.725,A -85,B 0,C 180,E1 -9174.496,E2 -9174.496} C_VEL
LIN {X 0,Y 439.636,Z 461.723,A -85,B 0,C 180,E1 -9178.168,E2 -9178.168} C_VEL
LIN {X 0,Y 439.766,Z 461.708,A -85,B 0,C 180,E1 -9180,E2 -9180} C_VEL
LIN {X 0,Y 439.657,Z 461.722,A -85,B 0,C 180,E1 -9182.749,E2 -9182.749} C_VEL
LIN {X 0,Y 439.621,Z 461.725,A -85,B 0,C 180,E1 -9186.425,E2 -9186.425} C_VEL
LIN {X 0,Y 439.502,Z 461.739,A -85,B 0,C 180,E1 -9189.202,E2 -9189.202} C_VEL
LIN {X 0,Y 439.468,Z 461.742,A -85,B 0,C 180,E1 -9192.938,E2 -9192.938} C_VEL
LIN {X 0,Y 439.45,Z 461.746,A -85,B 0,C 180,E1 -9196.349,E2 -9196.349} C_VEL
LIN {X 0,Y 439.405,Z 461.749,A -85,B 0,C 180,E1 -9199.626,E2 -9199.626} C_VEL
LIN {X 0,Y 439.367,Z 461.757,A -85,B 0,C 180,E1 -9202.576,E2 -9202.576} C_VEL
LIN {X 0,Y 439.407,Z 461.749,A -85,B 0,C 180,E1 -9205.585,E2 -9205.585} C_VEL
LIN {X 0,Y 439.42,Z 461.749,A -85,B 0,C 180,E1 -9208.674,E2 -9208.674} C_VEL
LIN {X 0,Y 439.373,Z 461.755,A -85,B 0,C 180,E1 -9212.031,E2 -9212.031} C_VEL
LIN {X 0,Y 439.399,Z 461.751,A -85,B 0,C 180,E1 -9215.341,E2 -9215.341} C_VEL
LIN {X 0,Y 439.385,Z 461.756,A -85,B 0,C 180,E1 -9218.595,E2 -9218.595} C_VEL
LIN {X 0,Y 439.392,Z 461.751,A -85,B 0,C 180,E1 -9221.257,E2 -9221.257} C_VEL
LIN {X 0,Y 439.409,Z 461.752,A -85,B 0,C 180,E1 -9224.729,E2 -9224.729} C_VEL
LIN {X 0,Y 439.399,Z 461.751,A -85,B 0,C 180,E1 -9227.796,E2 -9227.796} C_VEL
LIN {X 0,Y 439.433,Z 461.748,A -85,B 0,C 180,E1 -9230.228,E2 -9230.228} C_VEL
LIN {X 0,Y 439.38,Z 461.753,A -85,B 0,C 180,E1 -9233.713,E2 -9233.713} C_VEL
LIN {X 0,Y 439.376,Z 461.754,A -85,B 0,C 180,E1 -9237.054,E2 -9237.054} C_VEL
LIN {X 0,Y 439.386,Z 461.755,A -85,B 0,C 180,E1 -9240.274,E2 -9240.274} C_VEL
LIN {X 0,Y 439.432,Z 461.746,A -85,B 0,C 180,E1 -9243.396,E2 -9243.396} C_VEL
LIN {X 0,Y 439.391,Z 461.754,A -85,B 0,C 180,E1 -9246.43,E2 -9246.43} C_VEL
LIN {X 0,Y 439.392,Z 461.75,A -85,B 0,C 180,E1 -9249.397,E2 -9249.397} C_VEL
LIN {X 0,Y 439.43,Z 461.748,A -85,B 0,C 180,E1 -9252.31,E2 -9252.31} C_VEL
LIN {X 0,Y 439.452,Z 461.744,A -85,B 0,C 180,E1 -9255.174,E2 -9255.174} C_VEL
LIN {X 0,Y 439.488,Z 461.743,A -85,B 0,C 180,E1 -9258.001,E2 -9258.001} C_VEL
LIN {X 0,Y 439.538,Z 461.735,A -85,B 0,C 180,E1 -9261.726,E2 -9261.726} C_VEL
LIN {X 0,Y 439.614,Z 461.724,A -85,B 0,C 180,E1 -9264.496,E2 -9264.496} C_VEL
LIN {X 0,Y 439.64,Z 461.723,A -85,B 0,C 180,E1 -9268.168,E2 -9268.168} C_VEL
LIN {X 0,Y 439.768,Z 461.708,A -85,B 0,C 180,E1 -9270,E2 -9270} C_VEL
LIN {X 0,Y 439.614,Z 461.722,A -85,B 0,C 180,E1 -9270.99,E2 -9270.99} C_VEL
LIN {X 0,Y 438.905,Z 461.815,A -85,B 0,C 180,E1 -9271.754,E2 -9271.754} C_VEL
LIN {X 0,Y 435.93,Z 462.183,A -85,B 0,C 180,E1 -9272.993,E2 -9272.993} C_VEL
LIN {X 0,Y 433.478,Z 462.49,A -85,B 0,C 180,E1 -9273.993,E2 -9273.993} C_VEL
LIN {X 0,Y 432.504,Z 462.611,A -85,B 0,C 180,E1 -9274.768,E2 -9274.768} C_VEL
LIN {X 0,Y 432.468,Z 462.614,A -85,B 0,C 180,E1 -9275.03,E2 -9275.03} C_VEL
LIN {X 0,Y 432.544,Z 462.606,A -85,B 0,C 180,E1 -9277.632,E2 -9277.632} C_VEL
LIN {X 0,Y 432.397,Z 462.624,A -85,B 0,C 180,E1 -9281.247,E2 -9281.247} C_VEL
LIN {X 0,Y 432.379,Z 462.629,A -85,B 0,C 180,E1 -9284.112,E2 -9284.112} C_VEL
LIN {X 0,Y 432.402,Z 462.622,A -85,B 0,C 180,E1 -9287.012,E2 -9287.012} C_VEL
LIN {X 0,Y 432.344,Z 462.632,A -85,B 0,C 180,E1 -9289.96,E2 -9289.96} C_VEL
LIN {X 0,Y 432.324,Z 462.63,A -85,B 0,C 180,E1 -9292.964,E2 -9292.964} C_VEL
LIN {X 0,Y 432.369,Z 462.628,A -85,B 0,C 180,E1 -9296.032,E2 -9296.032} C_VEL
LIN {X 0,Y 432.348,Z 462.629,A -85,B 0,C 180,E1 -9299.187,E2 -9299.187} C_VEL
LIN {X 0,Y 432.327,Z 462.633,A -85,B 0,C 180,E1 -9302.443,E2 -9302.443} C_VEL
LIN {X 0,Y 432.348,Z 462.631,A -85,B 0,C 180,E1 -9305.632,E2 -9305.632} C_VEL
LIN {X 0,Y 432.355,Z 462.628,A -85,B 0,C 180,E1 -9308.716,E2 -9308.716} C_VEL
LIN {X 0,Y 432.337,Z 462.632,A -85,B 0,C 180,E1 -9311.797,E2 -9311.797} C_VEL
LIN {X 0,Y 432.337,Z 462.63,A -85,B 0,C 180,E1 -9314.347,E2 -9314.347} C_VEL
LIN {X 0,Y 432.324,Z 462.633,A -85,B 0,C 180,E1 -9317.016,E2 -9317.016} C_VEL
LIN {X 0,Y 432.337,Z 462.633,A -85,B 0,C 180,E1 -9319.821,E2 -9319.821} C_VEL
LIN {X 0,Y 432.3,Z 462.635,A -85,B 0,C 180,E1 -9323.021,E2 -9323.021} C_VEL
LIN {X 0,Y 432.128,Z 462.66,A -85,B 0,C 180,E1 -9326.043,E2 -9326.043} C_VEL
LIN {X 0,Y 431.824,Z 462.696,A -85,B 0,C 180,E1 -9328.613,E2 -9328.613} C_VEL
LIN {X 0,Y 431.614,Z 463.078,A -85,B 0,C 180,E1 -9330.758,E2 -9330.758} C_VEL
LIN {X 0,Y 431.612,Z 466.26,A -85,B 0,C 180,E1 -9333.918,E2 -9333.918} C_VEL
LIN {X 0,Y 431.499,Z 469.453,A -85,B 0,C 180,E1 -9336.989,E2 -9336.989} C_VEL
LIN {X 0,Y 431.424,Z 472.616,A -85,B 0,C 180,E1 -9339.995,E2 -9339.995} C_VEL
LIN {X 0,Y 431.407,Z 476.264,A -85,B 0,C 180,E1 -9343.387,E2 -9343.387} C_VEL
LIN {X 0,Y 431.395,Z 476.502,A -85,B 0,C 180,E1 -9343.604,E2 -9343.604} C_VEL
LIN {X 0,Y 434.797,Z 491.868,A -85,B 0,C 180,E1 -9344.291,E2 -9344.291} C_VEL
LIN {X 0,Y 435.562,Z 495.674,A -85,B 0,C 180,E1 -9344.499,E2 -9344.499} C_VEL
LIN {X 0,Y 435.132,Z 507.241,A -85,B 0,C 180,E1 -9345.143,E2 -9345.143} C_VEL
LIN {X 0,Y 434.561,Z 518.688,A -85,B 0,C 180,E1 -9345.96,E2 -9345.96} C_VEL
LIN {X 0,Y 433.98,Z 530.302,A -85,B 0,C 180,E1 -9347.015,E2 -9347.015} C_VEL
LIN {X 0,Y 433.371,Z 539.745,A -85,B 0,C 180,E1 -9348.067,E2 -9348.067} C_VEL
LIN {X 0,Y 432.886,Z 548.405,A -85,B 0,C 180,E1 -9349.239,E2 -9349.239} C_VEL
LIN {X 0,Y 432.391,Z 556.826,A -85,B 0,C 180,E1 -9350.646,E2 -9350.646} C_VEL
LIN {X 0,Y 431.957,Z 563.629,A -85,B 0,C 180,E1 -9352.051,E2 -9352.051} C_VEL
LIN {X 0,Y 431.788,Z 569.061,A -85,B 0,C 180,E1 -9353.458,E2 -9353.458} C_VEL
LIN {X 0,Y 431.487,Z 573.31,A -85,B 0,C 180,E1 -9354.86,E2 -9354.86} C_VEL
LIN {X 0,Y 431.474,Z 576.471,A -85,B 0,C 180,E1 -9356.264,E2 -9356.264} C_VEL
LIN {X 0,Y 431.403,Z 578.047,A -85,B 0,C 180,E1 -9357.198,E2 -9357.198} C_VEL
LIN {X 0,Y 431.334,Z 579.161,A -85,B 0,C 180,E1 -9358.132,E2 -9358.132} C_VEL
LIN {X 0,Y 431.293,Z 579.881,A -85,B 0,C 180,E1 -9359.066,E2 -9359.066} C_VEL
LIN {X 0,Y 431.278,Z 580.209,A -85,B 0,C 180,E1 -9360,E2 -9360} C_VEL
LIN {X 0,Y 431.31,Z 580.117,A -85,B 0,C 180,E1 -9360.933,E2 -9360.933} C_VEL
LIN {X 0,Y 431.393,Z 579.594,A -85,B 0,C 180,E1 -9361.867,E2 -9361.867} C_VEL
LIN {X 0,Y 431.515,Z 577.377,A -85,B 0,C 180,E1 -9363.735,E2 -9363.735} C_VEL
LIN {X 0,Y 431.571,Z 574.579,A -85,B 0,C 180,E1 -9365.138,E2 -9365.138} C_VEL
LIN {X 0,Y 431.864,Z 570.732,A -85,B 0,C 180,E1 -9366.541,E2 -9366.541} C_VEL
LIN {X 0,Y 432.104,Z 565.755,A -85,B 0,C 180,E1 -9367.946,E2 -9367.946} C_VEL
LIN {X 0,Y 432.573,Z 559.444,A -85,B 0,C 180,E1 -9369.35,E2 -9369.35} C_VEL
LIN {X 0,Y 433.09,Z 551.578,A -85,B 0,C 180,E1 -9370.755,E2 -9370.755} C_VEL
LIN {X 0,Y 433.65,Z 541.833,A -85,B 0,C 180,E1 -9372.162,E2 -9372.162} C_VEL
LIN {X 0,Y 434.512,Z 531.933,A -85,B 0,C 180,E1 -9373.298,E2 -9373.298} C_VEL
LIN {X 0,Y 435.132,Z 520.704,A -85,B 0,C 180,E1 -9374.354,E2 -9374.354} C_VEL
LIN {X 0,Y 435.768,Z 509.386,A -85,B 0,C 180,E1 -9375.193,E2 -9375.193} C_VEL
LIN {X 0,Y 436.334,Z 497.275,A -85,B 0,C 180,E1 -9375.892,E2 -9375.892} C_VEL
LIN {X 0,Y 434.434,Z 488.572,A -85,B 0,C 180,E1 -9376.394,E2 -9376.394} C_VEL
LIN {X 0,Y 431.754,Z 479.597,A -85,B 0,C 180,E1 -9376.885,E2 -9376.885} C_VEL
LIN {X 0,Y 431.837,Z 477.004,A -85,B 0,C 180,E1 -9379.985,E2 -9379.985} C_VEL
LIN {X 0,Y 431.973,Z 474.639,A -85,B 0,C 180,E1 -9382.984,E2 -9382.984} C_VEL
LIN {X 0,Y 432.174,Z 472.419,A -85,B 0,C 180,E1 -9386.045,E2 -9386.045} C_VEL
LIN {X 0,Y 432.384,Z 470.387,A -85,B 0,C 180,E1 -9389.184,E2 -9389.184} C_VEL
LIN {X 0,Y 432.722,Z 468.634,A -85,B 0,C 180,E1 -9392.409,E2 -9392.409} C_VEL
LIN {X 0,Y 432.883,Z 467.694,A -85,B 0,C 180,E1 -9394.627,E2 -9394.627} C_VEL
LIN {X 0,Y 432.985,Z 466.936,A -85,B 0,C 180,E1 -9397.312,E2 -9397.312} C_VEL
LIN {X 0,Y 433.039,Z 466.702,A -85,B 0,C 180,E1 -9400.48,E2 -9400.48} C_VEL
LIN {X 0,Y 433.126,Z 467.172,A -85,B 0,C 180,E1 -9403.098,E2 -9403.098} C_VEL
LIN {X 0,Y 433.373,Z 468.348,A -85,B 0,C 180,E1 -9405.786,E2 -9405.786} C_VEL
LIN {X 0,Y 433.718,Z 470.277,A -85,B 0,C 180,E1 -9408.366,E2 -9408.366} C_VEL
LIN {X 0,Y 434.179,Z 472.994,A -85,B 0,C 180,E1 -9410.984,E2 -9410.984} C_VEL
LIN {X 0,Y 434.483,Z 475.98,A -85,B 0,C 180,E1 -9413.238,E2 -9413.238} C_VEL
LIN {X 0,Y 434.488,Z 477.754,A -85,B 0,C 180,E1 -9414.386,E2 -9414.386} C_VEL
LIN {X 0,Y 434.051,Z 481.634,A -85,B 0,C 180,E1 -9416.597,E2 -9416.597} C_VEL
LIN {X 0,Y 433.429,Z 486.869,A -85,B 0,C 180,E1 -9419.248,E2 -9419.248} C_VEL
LIN {X 0,Y 432.753,Z 495,A -85,B 0,C 180,E1 -9422.953,E2 -9422.953} C_VEL
LIN {X 0,Y 432.289,Z 502.334,A -85,B 0,C 180,E1 -9426.018,E2 -9426.018} C_VEL
LIN {X 0,Y 431.997,Z 509.946,A -85,B 0,C 180,E1 -9429.028,E2 -9429.028} C_VEL
LIN {X 0,Y 431.683,Z 519.003,A -85,B 0,C 180,E1 -9432.471,E2 -9432.471} C_VEL
LIN {X 0,Y 431.687,Z 520.614,A -85,B 0,C 180,E1 -9433.069,E2 -9433.069} C_VEL
LIN {X 0,Y 433.932,Z 534.646,A -85,B 0,C 180,E1 -9433.66,E2 -9433.66} C_VEL
LIN {X 0,Y 435.189,Z 547.985,A -85,B 0,C 180,E1 -9434.366,E2 -9434.366} C_VEL
LIN {X 0,Y 434.684,Z 560.168,A -85,B 0,C 180,E1 -9435.127,E2 -9435.127} C_VEL
LIN {X 0,Y 433.952,Z 571.941,A -85,B 0,C 180,E1 -9436.054,E2 -9436.054} C_VEL
LIN {X 0,Y 433.234,Z 583.817,A -85,B 0,C 180,E1 -9437.23,E2 -9437.23} C_VEL
LIN {X 0,Y 432.703,Z 592.531,A -85,B 0,C 180,E1 -9438.286,E2 -9438.286} C_VEL
LIN {X 0,Y 432.177,Z 600.633,A -85,B 0,C 180,E1 -9439.458,E2 -9439.458} C_VEL
LIN {X 0,Y 431.775,Z 608.629,A -85,B 0,C 180,E1 -9440.868,E2 -9440.868} C_VEL
LIN {X 0,Y 431.548,Z 614.117,A -85,B 0,C 180,E1 -9442.043,E2 -9442.043} C_VEL
LIN {X 0,Y 431.359,Z 620.081,A -85,B 0,C 180,E1 -9443.646,E2 -9443.646} C_VEL
LIN {X 0,Y 431.291,Z 624.761,A -85,B 0,C 180,E1 -9445.326,E2 -9445.326} C_VEL
LIN {X 0,Y 431.245,Z 626.721,A -85,B 0,C 180,E1 -9446.262,E2 -9446.262} C_VEL
LIN {X 0,Y 431.326,Z 628.204,A -85,B 0,C 180,E1 -9447.198,E2 -9447.198} C_VEL
LIN {X 0,Y 431.287,Z 629.268,A -85,B 0,C 180,E1 -9448.132,E2 -9448.132} C_VEL
LIN {X 0,Y 431.276,Z 629.93,A -85,B 0,C 180,E1 -9449.066,E2 -9449.066} C_VEL
LIN {X 0,Y 431.277,Z 630.156,A -85,B 0,C 180,E1 -9450,E2 -9450} C_VEL
LIN {X 0,Y 431.289,Z 629.944,A -85,B 0,C 180,E1 -9450.934,E2 -9450.934} C_VEL
LIN {X 0,Y 431.285,Z 629.329,A -85,B 0,C 180,E1 -9451.868,E2 -9451.868} C_VEL
LIN {X 0,Y 431.318,Z 628.311,A -85,B 0,C 180,E1 -9452.802,E2 -9452.802} C_VEL
LIN {X 0,Y 431.238,Z 626.822,A -85,B 0,C 180,E1 -9453.738,E2 -9453.738} C_VEL
LIN {X 0,Y 431.352,Z 623.774,A -85,B 0,C 180,E1 -9455.141,E2 -9455.141} C_VEL
LIN {X 0,Y 431.376,Z 619.624,A -85,B 0,C 180,E1 -9456.548,E2 -9456.548} C_VEL
LIN {X 0,Y 431.603,Z 613.257,A -85,B 0,C 180,E1 -9458.191,E2 -9458.191} C_VEL
LIN {X 0,Y 431.908,Z 606.317,A -85,B 0,C 180,E1 -9459.601,E2 -9459.601} C_VEL
LIN {X 0,Y 432.38,Z 597.636,A -85,B 0,C 180,E1 -9461.01,E2 -9461.01} C_VEL
LIN {X 0,Y 432.903,Z 588.761,A -85,B 0,C 180,E1 -9462.184,E2 -9462.184} C_VEL
LIN {X 0,Y 433.568,Z 578.599,A -85,B 0,C 180,E1 -9463.285,E2 -9463.285} C_VEL
LIN {X 0,Y 434.17,Z 567.016,A -85,B 0,C 180,E1 -9464.291,E2 -9464.291} C_VEL
LIN {X 0,Y 434.831,Z 555.048,A -85,B 0,C 180,E1 -9465.107,E2 -9465.107} C_VEL
LIN {X 0,Y 435.119,Z 548.814,A -85,B 0,C 180,E1 -9465.456,E2 -9465.456} C_VEL
LIN {X 0,Y 433.532,Z 535.755,A -85,B 0,C 180,E1 -9466.093,E2 -9466.093} C_VEL
LIN {X 0,Y 431.739,Z 523.284,A -85,B 0,C 180,E1 -9466.547,E2 -9466.547} C_VEL
LIN {X 0,Y 431.993,Z 514.289,A -85,B 0,C 180,E1 -9469.977,E2 -9469.977} C_VEL
LIN {X 0,Y 432.403,Z 505.324,A -85,B 0,C 180,E1 -9473.466,E2 -9473.466} C_VEL
LIN {X 0,Y 432.926,Z 496.328,A -85,B 0,C 180,E1 -9477.036,E2 -9477.036} C_VEL
LIN {X 0,Y 433.335,Z 489.911,A -85,B 0,C 180,E1 -9479.647,E2 -9479.647} C_VEL
LIN {X 0,Y 433.848,Z 482.822,A -85,B 0,C 180,E1 -9482.61,E2 -9482.61} C_VEL
LIN {X 0,Y 434.332,Z 475.793,A -85,B 0,C 180,E1 -9485.628,E2 -9485.628} C_VEL
LIN {X 0,Y 433.985,Z 471.727,A -85,B 0,C 180,E1 -9487.485,E2 -9487.485} C_VEL
LIN {X 0,Y 432.871,Z 465.426,A -85,B 0,C 180,E1 -9490.499,E2 -9490.499} C_VEL
LIN {X 0,Y 432.367,Z 462.63,A -85,B 0,C 180,E1 -9491.95,E2 -9491.95} C_VEL
LIN {X 0,Y 432.38,Z 462.627,A -85,B 0,C 180,E1 -9495.659,E2 -9495.659} C_VEL
LIN {X 0,Y 432.369,Z 462.628,A -85,B 0,C 180,E1 -9498.393,E2 -9498.393} C_VEL
LIN {X 0,Y 432.337,Z 462.629,A -85,B 0,C 180,E1 -9501.85,E2 -9501.85} C_VEL
LIN {X 0,Y 432.341,Z 462.631,A -85,B 0,C 180,E1 -9505.323,E2 -9505.323} C_VEL
LIN {X 0,Y 432.323,Z 462.636,A -85,B 0,C 180,E1 -9508.654,E2 -9508.654} C_VEL
LIN {X 0,Y 432.384,Z 462.626,A -85,B 0,C 180,E1 -9511.877,E2 -9511.877} C_VEL
LIN {X 0,Y 432.353,Z 462.63,A -85,B 0,C 180,E1 -9514.999,E2 -9514.999} C_VEL
LIN {X 0,Y 432.359,Z 462.629,A -85,B 0,C 180,E1 -9518.046,E2 -9518.046} C_VEL
LIN {X 0,Y 432.388,Z 462.626,A -85,B 0,C 180,E1 -9521.03,E2 -9521.03} C_VEL
LIN {X 0,Y 432.433,Z 462.619,A -85,B 0,C 180,E1 -9523.961,E2 -9523.961} C_VEL
LIN {X 0,Y 432.461,Z 462.616,A -85,B 0,C 180,E1 -9527.804,E2 -9527.804} C_VEL
LIN {X 0,Y 432.494,Z 462.611,A -85,B 0,C 180,E1 -9531.59,E2 -9531.59} C_VEL
LIN {X 0,Y 432.599,Z 462.599,A -85,B 0,C 180,E1 -9534.406,E2 -9534.406} C_VEL
LIN {X 0,Y 432.606,Z 462.599,A -85,B 0,C 180,E1 -9538.138,E2 -9538.138} C_VEL
LIN {X 0,Y 432.736,Z 462.583,A -85,B 0,C 180,E1 -9540,E2 -9540} C_VEL
LIN {X 0,Y 432.606,Z 462.6,A -85,B 0,C 180,E1 -9542.794,E2 -9542.794} C_VEL
LIN {X 0,Y 432.575,Z 462.603,A -85,B 0,C 180,E1 -9546.53,E2 -9546.53} C_VEL
LIN {X 0,Y 432.445,Z 462.617,A -85,B 0,C 180,E1 -9549.353,E2 -9549.353} C_VEL
LIN {X 0,Y 432.433,Z 462.619,A -85,B 0,C 180,E1 -9552.804,E2 -9552.804} C_VEL
LIN {X 0,Y 432.415,Z 462.623,A -85,B 0,C 180,E1 -9556.479,E2 -9556.479} C_VEL
LIN {X 0,Y 432.342,Z 462.631,A -85,B 0,C 180,E1 -9559.961,E2 -9559.961} C_VEL
LIN {X 0,Y 432.321,Z 462.634,A -85,B 0,C 180,E1 -9562.964,E2 -9562.964} C_VEL
LIN {X 0,Y 432.367,Z 462.628,A -85,B 0,C 180,E1 -9566.033,E2 -9566.033} C_VEL
LIN {X 0,Y 432.346,Z 462.63,A -85,B 0,C 180,E1 -9569.188,E2 -9569.188} C_VEL
LIN {X 0,Y 432.326,Z 462.636,A -85,B 0,C 180,E1 -9572.443,E2 -9572.443} C_VEL
LIN {X 0,Y 432.348,Z 462.63,A -85,B 0,C 180,E1 -9575.632,E2 -9575.632} C_VEL
LIN {X 0,Y 432.347,Z 462.631,A -85,B 0,C 180,E1 -9578.715,E2 -9578.715} C_VEL
LIN {X 0,Y 432.338,Z 462.632,A -85,B 0,C 180,E1 -9581.797,E2 -9581.797} C_VEL
LIN {X 0,Y 432.344,Z 462.631,A -85,B 0,C 180,E1 -9584.347,E2 -9584.347} C_VEL
LIN {X 0,Y 432.326,Z 462.631,A -85,B 0,C 180,E1 -9587.016,E2 -9587.016} C_VEL
LIN {X 0,Y 432.34,Z 462.633,A -85,B 0,C 180,E1 -9589.82,E2 -9589.82} C_VEL
LIN {X 0,Y 432.319,Z 462.633,A -85,B 0,C 180,E1 -9593.023,E2 -9593.023} C_VEL
LIN {X 0,Y 432.363,Z 462.631,A -85,B 0,C 180,E1 -9595.997,E2 -9595.997} C_VEL
LIN {X 0,Y 432.351,Z 462.63,A -85,B 0,C 180,E1 -9599.49,E2 -9599.49} C_VEL
LIN {X 0,Y 432.395,Z 462.623,A -85,B 0,C 180,E1 -9602.928,E2 -9602.928} C_VEL
LIN {X 0,Y 432.375,Z 462.627,A -85,B 0,C 180,E1 -9606.024,E2 -9606.024} C_VEL
LIN {X 0,Y 432.354,Z 462.627,A -85,B 0,C 180,E1 -9609.046,E2 -9609.046} C_VEL
LIN {X 0,Y 432.378,Z 462.628,A -85,B 0,C 180,E1 -9612.011,E2 -9612.011} C_VEL
LIN {X 0,Y 432.4,Z 462.623,A -85,B 0,C 180,E1 -9614.927,E2 -9614.927} C_VEL
LIN {X 0,Y 432.464,Z 462.618,A -85,B 0,C 180,E1 -9617.804,E2 -9617.804} C_VEL
LIN {X 0,Y 432.487,Z 462.613,A -85,B 0,C 180,E1 -9621.59,E2 -9621.59} C_VEL
LIN {X 0,Y 432.59,Z 462.6,A -85,B 0,C 180,E1 -9624.406,E2 -9624.406} C_VEL
LIN {X 0,Y 432.61,Z 462.599,A -85,B 0,C 180,E1 -9628.138,E2 -9628.138} C_VEL
LIN {X 0,Y 432.737,Z 462.584,A -85,B 0,C 180,E1 -9630,E2 -9630} C_VEL
LIN {X 0,Y 432.597,Z 462.598,A -85,B 0,C 180,E1 -9632.794,E2 -9632.794} C_VEL
LIN {X 0,Y 432.468,Z 462.614,A -85,B 0,C 180,E1 -9635.03,E2 -9635.03} C_VEL
LIN {X 0,Y 431.907,Z 462.686,A -85,B 0,C 180,E1 -9635.809,E2 -9635.809} C_VEL
LIN {X 0,Y 429.059,Z 463.038,A -85,B 0,C 180,E1 -9637.073,E2 -9637.073} C_VEL
LIN {X 0,Y 426.573,Z 463.352,A -85,B 0,C 180,E1 -9638.093,E2 -9638.093} C_VEL
LIN {X 0,Y 425.494,Z 463.482,A -85,B 0,C 180,E1 -9638.883,E2 -9638.883} C_VEL
LIN {X 0,Y 425.404,Z 463.493,A -85,B 0,C 180,E1 -9639.151,E2 -9639.151} C_VEL
LIN {X 0,Y 425.398,Z 463.495,A -85,B 0,C 180,E1 -9642.904,E2 -9642.904} C_VEL
LIN {X 0,Y 425.366,Z 463.499,A -85,B 0,C 180,E1 -9646.605,E2 -9646.605} C_VEL
LIN {X 0,Y 425.333,Z 463.505,A -85,B 0,C 180,E1 -9649.636,E2 -9649.636} C_VEL
LIN {X 0,Y 425.312,Z 463.505,A -85,B 0,C 180,E1 -9653.365,E2 -9653.365} C_VEL
LIN {X 0,Y 425.352,Z 463.501,A -85,B 0,C 180,E1 -9656.844,E2 -9656.844} C_VEL
LIN {X 0,Y 425.295,Z 463.51,A -85,B 0,C 180,E1 -9659.719,E2 -9659.719} C_VEL
LIN {X 0,Y 425.286,Z 463.509,A -85,B 0,C 180,E1 -9663.048,E2 -9663.048} C_VEL
LIN {X 0,Y 425.287,Z 463.512,A -85,B 0,C 180,E1 -9665.929,E2 -9665.929} C_VEL
LIN {X 0,Y 425.304,Z 463.507,A -85,B 0,C 180,E1 -9669.044,E2 -9669.044} C_VEL
LIN {X 0,Y 425.278,Z 463.51,A -85,B 0,C 180,E1 -9672.653,E2 -9672.653} C_VEL
LIN {X 0,Y 425.265,Z 463.513,A -85,B 0,C 180,E1 -9676.044,E2 -9676.044} C_VEL
LIN {X 0,Y 425.278,Z 463.51,A -85,B 0,C 180,E1 -9678.621,E2 -9678.621} C_VEL
LIN {X 0,Y 425.309,Z 463.506,A -85,B 0,C 180,E1 -9681.102,E2 -9681.102} C_VEL
LIN {X 0,Y 425.22,Z 463.518,A -85,B 0,C 180,E1 -9684.083,E2 -9684.083} C_VEL
LIN {X 0,Y 424.949,Z 463.552,A -85,B 0,C 180,E1 -9686.922,E2 -9686.922} C_VEL
LIN {X 0,Y 424.605,Z 463.6,A -85,B 0,C 180,E1 -9690.227,E2 -9690.227} C_VEL
LIN {X 0,Y 424.566,Z 464.317,A -85,B 0,C 180,E1 -9691.322,E2 -9691.322} C_VEL
LIN {X 0,Y 424.495,Z 467.526,A -85,B 0,C 180,E1 -9694.503,E2 -9694.503} C_VEL
LIN {X 0,Y 424.398,Z 471.147,A -85,B 0,C 180,E1 -9698.027,E2 -9698.027} C_VEL
LIN {X 0,Y 424.375,Z 474.012,A -85,B 0,C 180,E1 -9700.73,E2 -9700.73} C_VEL
LIN {X 0,Y 424.333,Z 476.852,A -85,B 0,C 180,E1 -9703.376,E2 -9703.376} C_VEL
LIN {X 0,Y 427.627,Z 491.588,A -85,B 0,C 180,E1 -9704.036,E2 -9704.036} C_VEL
LIN {X 0,Y 428.642,Z 497.612,A -85,B 0,C 180,E1 -9704.362,E2 -9704.362} C_VEL
LIN {X 0,Y 428.064,Z 510.522,A -85,B 0,C 180,E1 -9705.135,E2 -9705.135} C_VEL
LIN {X 0,Y 427.44,Z 522.463,A -85,B 0,C 180,E1 -9706.061,E2 -9706.061} C_VEL
LIN {X 0,Y 426.807,Z 533.619,A -85,B 0,C 180,E1 -9707.156,E2 -9707.156} C_VEL
LIN {X 0,Y 426.191,Z 543.428,A -85,B 0,C 180,E1 -9708.346,E2 -9708.346} C_VEL
LIN {X 0,Y 425.68,Z 551.508,A -85,B 0,C 180,E1 -9709.536,E2 -9709.536} C_VEL
LIN {X 0,Y 425.194,Z 559.451,A -85,B 0,C 180,E1 -9710.966,E2 -9710.966} C_VEL
LIN {X 0,Y 424.829,Z 565.801,A -85,B 0,C 180,E1 -9712.395,E2 -9712.395} C_VEL
LIN {X 0,Y 424.662,Z 570.856,A -85,B 0,C 180,E1 -9713.824,E2 -9713.824} C_VEL
LIN {X 0,Y 424.399,Z 574.773,A -85,B 0,C 180,E1 -9715.25,E2 -9715.25} C_VEL
LIN {X 0,Y 424.388,Z 576.797,A -85,B 0,C 180,E1 -9716.202,E2 -9716.202} C_VEL
LIN {X 0,Y 424.335,Z 578.402,A -85,B 0,C 180,E1 -9717.152,E2 -9717.152} C_VEL
LIN {X 0,Y 424.255,Z 579.542,A -85,B 0,C 180,E1 -9718.101,E2 -9718.101} C_VEL
LIN {X 0,Y 424.203,Z 580.628,A -85,B 0,C 180,E1 -9720,E2 -9720} C_VEL
LIN {X 0,Y 424.253,Z 580.567,A -85,B 0,C 180,E1 -9720.949,E2 -9720.949} C_VEL
LIN {X 0,Y 424.323,Z 580.063,A -85,B 0,C 180,E1 -9721.898,E2 -9721.898} C_VEL
LIN {X 0,Y 424.465,Z 577.876,A -85,B 0,C 180,E1 -9723.797,E2 -9723.797} C_VEL
LIN {X 0,Y 424.525,Z 575.104,A -85,B 0,C 180,E1 -9725.224,E2 -9725.224} C_VEL
LIN {X 0,Y 424.832,Z 571.282,A -85,B 0,C 180,E1 -9726.65,E2 -9726.65} C_VEL
LIN {X 0,Y 425.115,Z 566.329,A -85,B 0,C 180,E1 -9728.078,E2 -9728.078} C_VEL
LIN {X 0,Y 425.61,Z 560.083,A -85,B 0,C 180,E1 -9729.505,E2 -9729.505} C_VEL
LIN {X 0,Y 426.156,Z 552.302,A -85,B 0,C 180,E1 -9730.932,E2 -9730.932} C_VEL
LIN {X 0,Y 426.761,Z 542.668,A -85,B 0,C 180,E1 -9732.362,E2 -9732.362} C_VEL
LIN {X 0,Y 427.673,Z 532.879,A -85,B 0,C 180,E1 -9733.511,E2 -9733.511} C_VEL
LIN {X 0,Y 428.331,Z 521.711,A -85,B 0,C 180,E1 -9734.587,E2 -9734.587} C_VEL
LIN {X 0,Y 429.01,Z 510.601,A -85,B 0,C 180,E1 -9735.439,E2 -9735.439} C_VEL
LIN {X 0,Y 429.547,Z 497.756,A -85,B 0,C 180,E1 -9736.21,E2 -9736.21} C_VEL
LIN {X 0,Y 426.791,Z 486.728,A -85,B 0,C 180,E1 -9736.882,E2 -9736.882} C_VEL
LIN {X 0,Y 424.71,Z 480.202,A -85,B 0,C 180,E1 -9737.26,E2 -9737.26} C_VEL
LIN {X 0,Y 424.814,Z 477.694,A -85,B 0,C 180,E1 -9740.329,E2 -9740.329} C_VEL
LIN {X 0,Y 424.992,Z 475.383,A -85,B 0,C 180,E1 -9743.383,E2 -9743.383} C_VEL
LIN {X 0,Y 425.231,Z 473.003,A -85,B 0,C 180,E1 -9746.812,E2 -9746.812} C_VEL
LIN {X 0,Y 425.409,Z 471.275,A -85,B 0,C 180,E1 -9749.71,E2 -9749.71} C_VEL
LIN {X 0,Y 425.767,Z 469.63,A -85,B 0,C 180,E1 -9753.006,E2 -9753.006} C_VEL
LIN {X 0,Y 425.945,Z 468.812,A -85,B 0,C 180,E1 -9755.274,E2 -9755.274} C_VEL
LIN {X 0,Y 426.044,Z 468.28,A -85,B 0,C 180,E1 -9757.645,E2 -9757.645} C_VEL
LIN {X 0,Y 426.087,Z 468.205,A -85,B 0,C 180,E1 -9760.647,E2 -9760.647} C_VEL
LIN {X 0,Y 426.26,Z 468.959,A -85,B 0,C 180,E1 -9763.827,E2 -9763.827} C_VEL
LIN {X 0,Y 426.528,Z 470.359,A -85,B 0,C 180,E1 -9766.469,E2 -9766.469} C_VEL
LIN {X 0,Y 426.913,Z 472.626,A -85,B 0,C 180,E1 -9769.224,E2 -9769.224} C_VEL
LIN {X 0,Y 427.455,Z 475.891,A -85,B 0,C 180,E1 -9772.11,E2 -9772.11} C_VEL
LIN {X 0,Y 427.532,Z 478.138,A -85,B 0,C 180,E1 -9773.716,E2 -9773.716} C_VEL
LIN {X 0,Y 427.205,Z 481.868,A -85,B 0,C 180,E1 -9775.99,E2 -9775.99} C_VEL
LIN {X 0,Y 426.401,Z 488.118,A -85,B 0,C 180,E1 -9779.273,E2 -9779.273} C_VEL
LIN {X 0,Y 425.831,Z 494.948,A -85,B 0,C 180,E1 -9782.476,E2 -9782.476} C_VEL
LIN {X 0,Y 425.313,Z 502.166,A -85,B 0,C 180,E1 -9785.6,E2 -9785.6} C_VEL
LIN {X 0,Y 424.925,Z 510.958,A -85,B 0,C 180,E1 -9789.17,E2 -9789.17} C_VEL
LIN {X 0,Y 424.622,Z 520.072,A -85,B 0,C 180,E1 -9792.696,E2 -9792.696} C_VEL
LIN {X 0,Y 427.048,Z 534.433,A -85,B 0,C 180,E1 -9793.337,E2 -9793.337} C_VEL
LIN {X 0,Y 428.273,Z 548.39,A -85,B 0,C 180,E1 -9794.107,E2 -9794.107} C_VEL
LIN {X 0,Y 428.271,Z 553.302,A -85,B 0,C 180,E1 -9794.412,E2 -9794.412} C_VEL
LIN {X 0,Y 427.546,Z 564.969,A -85,B 0,C 180,E1 -9795.239,E2 -9795.239} C_VEL
LIN {X 0,Y 426.724,Z 576.765,A -85,B 0,C 180,E1 -9796.286,E2 -9796.286} C_VEL
LIN {X 0,Y 425.984,Z 586.687,A -85,B 0,C 180,E1 -9797.373,E2 -9797.373} C_VEL
LIN {X 0,Y 425.514,Z 595.677,A -85,B 0,C 180,E1 -9798.568,E2 -9798.568} C_VEL
LIN {X 0,Y 424.927,Z 604.548,A -85,B 0,C 180,E1 -9799.999,E2 -9799.999} C_VEL
LIN {X 0,Y 424.609,Z 611.683,A -85,B 0,C 180,E1 -9801.433,E2 -9801.433} C_VEL
LIN {X 0,Y 424.34,Z 617.431,A -85,B 0,C 180,E1 -9802.864,E2 -9802.864} C_VEL
LIN {X 0,Y 424.206,Z 621.965,A -85,B 0,C 180,E1 -9804.295,E2 -9804.295} C_VEL
LIN {X 0,Y 424.221,Z 624.384,A -85,B 0,C 180,E1 -9805.248,E2 -9805.248} C_VEL
LIN {X 0,Y 424.152,Z 626.327,A -85,B 0,C 180,E1 -9806.2,E2 -9806.2} C_VEL
LIN {X 0,Y 424.235,Z 627.805,A -85,B 0,C 180,E1 -9807.151,E2 -9807.151} C_VEL
LIN {X 0,Y 424.209,Z 628.866,A -85,B 0,C 180,E1 -9808.101,E2 -9808.101} C_VEL
LIN {X 0,Y 424.19,Z 629.522,A -85,B 0,C 180,E1 -9809.051,E2 -9809.051} C_VEL
LIN {X 0,Y 424.218,Z 629.731,A -85,B 0,C 180,E1 -9810,E2 -9810} C_VEL
LIN {X 0,Y 424.202,Z 629.51,A -85,B 0,C 180,E1 -9810.949,E2 -9810.949} C_VEL
LIN {X 0,Y 424.207,Z 628.885,A -85,B 0,C 180,E1 -9811.899,E2 -9811.899} C_VEL
LIN {X 0,Y 424.246,Z 627.854,A -85,B 0,C 180,E1 -9812.849,E2 -9812.849} C_VEL
LIN {X 0,Y 424.147,Z 626.34,A -85,B 0,C 180,E1 -9813.8,E2 -9813.8} C_VEL
LIN {X 0,Y 424.258,Z 623.262,A -85,B 0,C 180,E1 -9815.227,E2 -9815.227} C_VEL
LIN {X 0,Y 424.299,Z 619.078,A -85,B 0,C 180,E1 -9816.658,E2 -9816.658} C_VEL
LIN {X 0,Y 424.53,Z 612.673,A -85,B 0,C 180,E1 -9818.329,E2 -9818.329} C_VEL
LIN {X 0,Y 424.867,Z 605.687,A -85,B 0,C 180,E1 -9819.762,E2 -9819.762} C_VEL
LIN {X 0,Y 425.374,Z 596.936,A -85,B 0,C 180,E1 -9821.194,E2 -9821.194} C_VEL
LIN {X 0,Y 425.887,Z 588,A -85,B 0,C 180,E1 -9822.388,E2 -9822.388} C_VEL
LIN {X 0,Y 426.562,Z 578.129,A -85,B 0,C 180,E1 -9823.47,E2 -9823.47} C_VEL
LIN {X 0,Y 427.15,Z 567.608,A -85,B 0,C 180,E1 -9824.41,E2 -9824.41} C_VEL
LIN {X 0,Y 427.834,Z 555.897,A -85,B 0,C 180,E1 -9825.238,E2 -9825.238} C_VEL
LIN {X 0,Y 428.012,Z 548.741,A -85,B 0,C 180,E1 -9825.659,E2 -9825.659} C_VEL
LIN {X 0,Y 426.494,Z 535.801,A -85,B 0,C 180,E1 -9826.309,E2 -9826.309} C_VEL
LIN {X 0,Y 424.654,Z 522.998,A -85,B 0,C 180,E1 -9826.783,E2 -9826.783} C_VEL
LIN {X 0,Y 424.942,Z 513.913,A -85,B 0,C 180,E1 -9830.323,E2 -9830.323} C_VEL
LIN {X 0,Y 425.367,Z 504.939,A -85,B 0,C 180,E1 -9833.878,E2 -9833.878} C_VEL
LIN {X 0,Y 425.861,Z 497.297,A -85,B 0,C 180,E1 -9836.98,E2 -9836.98} C_VEL
LIN {X 0,Y 426.286,Z 490.876,A -85,B 0,C 180,E1 -9839.643,E2 -9839.643} C_VEL
LIN {X 0,Y 426.871,Z 483.184,A -85,B 0,C 180,E1 -9842.909,E2 -9842.909} C_VEL
LIN {X 0,Y 427.339,Z 476.791,A -85,B 0,C 180,E1 -9845.718,E2 -9845.718} C_VEL
LIN {X 0,Y 426.892,Z 472.329,A -85,B 0,C 180,E1 -9847.793,E2 -9847.793} C_VEL
LIN {X 0,Y 425.872,Z 466.547,A -85,B 0,C 180,E1 -9850.613,E2 -9850.613} C_VEL
LIN {X 0,Y 425.341,Z 463.505,A -85,B 0,C 180,E1 -9852.263,E2 -9852.263} C_VEL
LIN {X 0,Y 425.336,Z 463.506,A -85,B 0,C 180,E1 -9856.054,E2 -9856.054} C_VEL
LIN {X 0,Y 425.303,Z 463.508,A -85,B 0,C 180,E1 -9858.625,E2 -9858.625} C_VEL
LIN {X 0,Y 425.303,Z 463.507,A -85,B 0,C 180,E1 -9861.102,E2 -9861.102} C_VEL
LIN {X 0,Y 425.3,Z 463.509,A -85,B 0,C 180,E1 -9864.664,E2 -9864.664} C_VEL
LIN {X 0,Y 425.266,Z 463.511,A -85,B 0,C 180,E1 -9868.073,E2 -9868.073} C_VEL
LIN {X 0,Y 425.333,Z 463.504,A -85,B 0,C 180,E1 -9871.368,E2 -9871.368} C_VEL
LIN {X 0,Y 425.297,Z 463.51,A -85,B 0,C 180,E1 -9874.555,E2 -9874.555} C_VEL
LIN {X 0,Y 425.289,Z 463.508,A -85,B 0,C 180,E1 -9877.661,E2 -9877.661} C_VEL
LIN {X 0,Y 425.364,Z 463.502,A -85,B 0,C 180,E1 -9880.704,E2 -9880.704} C_VEL
LIN {X 0,Y 425.39,Z 463.495,A -85,B 0,C 180,E1 -9883.688,E2 -9883.688} C_VEL
LIN {X 0,Y 425.414,Z 463.493,A -85,B 0,C 180,E1 -9887.598,E2 -9887.598} C_VEL
LIN {X 0,Y 425.444,Z 463.489,A -85,B 0,C 180,E1 -9891.45,E2 -9891.45} C_VEL
LIN {X 0,Y 425.556,Z 463.477,A -85,B 0,C 180,E1 -9894.313,E2 -9894.313} C_VEL
LIN {X 0,Y 425.575,Z 463.474,A -85,B 0,C 180,E1 -9898.107,E2 -9898.107} C_VEL
LIN {X 0,Y 425.706,Z 463.459,A -85,B 0,C 180,E1 -9900,E2 -9900} C_VEL
LIN {X 0,Y 425.558,Z 463.477,A -85,B 0,C 180,E1 -9902.84,E2 -9902.84} C_VEL
LIN {X 0,Y 425.533,Z 463.48,A -85,B 0,C 180,E1 -9906.639,E2 -9906.639} C_VEL
LIN {X 0,Y 425.404,Z 463.494,A -85,B 0,C 180,E1 -9909.51,E2 -9909.51} C_VEL
LIN {X 0,Y 425.396,Z 463.496,A -85,B 0,C 180,E1 -9912.904,E2 -9912.904} C_VEL
LIN {X 0,Y 425.364,Z 463.502,A -85,B 0,C 180,E1 -9916.605,E2 -9916.605} C_VEL
LIN {X 0,Y 425.331,Z 463.502,A -85,B 0,C 180,E1 -9919.636,E2 -9919.636} C_VEL
LIN {X 0,Y 425.309,Z 463.506,A -85,B 0,C 180,E1 -9923.365,E2 -9923.365} C_VEL
LIN {X 0,Y 425.351,Z 463.501,A -85,B 0,C 180,E1 -9926.845,E2 -9926.845} C_VEL
LIN {X 0,Y 425.294,Z 463.509,A -85,B 0,C 180,E1 -9929.72,E2 -9929.72} C_VEL
LIN {X 0,Y 425.285,Z 463.507,A -85,B 0,C 180,E1 -9933.048,E2 -9933.048} C_VEL
LIN {X 0,Y 425.287,Z 463.512,A -85,B 0,C 180,E1 -9935.929,E2 -9935.929} C_VEL
LIN {X 0,Y 425.293,Z 463.508,A -85,B 0,C 180,E1 -9939.042,E2 -9939.042} C_VEL
LIN {X 0,Y 425.281,Z 463.511,A -85,B 0,C 180,E1 -9942.653,E2 -9942.653} C_VEL
LIN {X 0,Y 425.266,Z 463.513,A -85,B 0,C 180,E1 -9946.045,E2 -9946.045} C_VEL
LIN {X 0,Y 425.278,Z 463.51,A -85,B 0,C 180,E1 -9948.622,E2 -9948.622} C_VEL
LIN {X 0,Y 425.316,Z 463.505,A -85,B 0,C 180,E1 -9951.103,E2 -9951.103} C_VEL
LIN {X 0,Y 425.304,Z 463.507,A -85,B 0,C 180,E1 -9954.665,E2 -9954.665} C_VEL
LIN {X 0,Y 425.269,Z 463.513,A -85,B 0,C 180,E1 -9958.073,E2 -9958.073} C_VEL
LIN {X 0,Y 425.335,Z 463.502,A -85,B 0,C 180,E1 -9961.368,E2 -9961.368} C_VEL
LIN {X 0,Y 425.3,Z 463.508,A -85,B 0,C 180,E1 -9964.555,E2 -9964.555} C_VEL
LIN {X 0,Y 425.292,Z 463.509,A -85,B 0,C 180,E1 -9967.662,E2 -9967.662} C_VEL
LIN {X 0,Y 425.365,Z 463.499,A -85,B 0,C 180,E1 -9970.704,E2 -9970.704} C_VEL
LIN {X 0,Y 425.392,Z 463.497,A -85,B 0,C 180,E1 -9973.688,E2 -9973.688} C_VEL
LIN {X 0,Y 425.417,Z 463.493,A -85,B 0,C 180,E1 -9977.598,E2 -9977.598} C_VEL
LIN {X 0,Y 425.441,Z 463.491,A -85,B 0,C 180,E1 -9981.45,E2 -9981.45} C_VEL
LIN {X 0,Y 425.545,Z 463.478,A -85,B 0,C 180,E1 -9984.313,E2 -9984.313} C_VEL
LIN {X 0,Y 425.579,Z 463.474,A -85,B 0,C 180,E1 -9988.107,E2 -9988.107} C_VEL
LIN {X 0,Y 425.707,Z 463.459,A -85,B 0,C 180,E1 -9990,E2 -9990} C_VEL
LIN {X 0,Y 425.55,Z 463.476,A -85,B 0,C 180,E1 -9992.84,E2 -9992.84} C_VEL
LIN {X 0,Y 425.556,Z 463.477,A -85,B 0,C 180,E1 -9995.687,E2 -9995.687} C_VEL
LIN {X 0,Y 425.44,Z 463.489,A -85,B 0,C 180,E1 -9998.55,E2 -9998.55} C_VEL
LIN {X 0,Y 425.404,Z 463.493,A -85,B 0,C 180,E1 -9999.151,E2 -9999.151} C_VEL
LIN {X 0,Y 424.735,Z 463.58,A -85,B 0,C 180,E1 -9999.94,E2 -9999.94} C_VEL
LIN {X 0,Y 421.889,Z 463.933,A -85,B 0,C 180,E1 -10001.224,E2 -10001.224} C_VEL
LIN {X 0,Y 419.472,Z 464.236,A -85,B 0,C 180,E1 -10002.26,E2 -10002.26} C_VEL
LIN {X 0,Y 418.421,Z 464.364,A -85,B 0,C 180,E1 -10003.061,E2 -10003.061} C_VEL
LIN {X 0,Y 418.327,Z 464.376,A -85,B 0,C 180,E1 -10003.332,E2 -10003.332} C_VEL
LIN {X 0,Y 418.318,Z 464.376,A -85,B 0,C 180,E1 -10006.736,E2 -10006.736} C_VEL
LIN {X 0,Y 418.276,Z 464.384,A -85,B 0,C 180,E1 -10009.79,E2 -10009.79} C_VEL
LIN {X 0,Y 418.243,Z 464.384,A -85,B 0,C 180,E1 -10012.736,E2 -10012.736} C_VEL
LIN {X 0,Y 418.275,Z 464.384,A -85,B 0,C 180,E1 -10015.904,E2 -10015.904} C_VEL
LIN {X 0,Y 418.269,Z 464.383,A -85,B 0,C 180,E1 -10019.162,E2 -10019.162} C_VEL
LIN {X 0,Y 418.262,Z 464.384,A -85,B 0,C 180,E1 -10022.844,E2 -10022.844} C_VEL
LIN {X 0,Y 418.25,Z 464.386,A -85,B 0,C 180,E1 -10026.238,E2 -10026.238} C_VEL
LIN {X 0,Y 418.256,Z 464.387,A -85,B 0,C 180,E1 -10029.682,E2 -10029.682} C_VEL
LIN {X 0,Y 418.233,Z 464.388,A -85,B 0,C 180,E1 -10032.321,E2 -10032.321} C_VEL
LIN {X 0,Y 418.239,Z 464.386,A -85,B 0,C 180,E1 -10035.109,E2 -10035.109} C_VEL
LIN {X 0,Y 418.244,Z 464.388,A -85,B 0,C 180,E1 -10037.767,E2 -10037.767} C_VEL
LIN {X 0,Y 418.256,Z 464.384,A -85,B 0,C 180,E1 -10040.619,E2 -10040.619} C_VEL
LIN {X 0,Y 418.192,Z 464.394,A -85,B 0,C 180,E1 -10043.97,E2 -10043.97} C_VEL
LIN {X 0,Y 417.966,Z 464.422,A -85,B 0,C 180,E1 -10046.297,E2 -10046.297} C_VEL
LIN {X 0,Y 417.607,Z 464.47,A -85,B 0,C 180,E1 -10049.676,E2 -10049.676} C_VEL
LIN {X 0,Y 417.506,Z 464.484,A -85,B 0,C 180,E1 -10050.78,E2 -10050.78} C_VEL
LIN {X 0,Y 417.428,Z 467.716,A -85,B 0,C 180,E1 -10054.039,E2 -10054.039} C_VEL
LIN {X 0,Y 417.318,Z 470.941,A -85,B 0,C 180,E1 -10057.211,E2 -10057.211} C_VEL
LIN {X 0,Y 417.307,Z 474.467,A -85,B 0,C 180,E1 -10060.582,E2 -10060.582} C_VEL
LIN {X 0,Y 417.263,Z 477.201,A -85,B 0,C 180,E1 -10063.141,E2 -10063.141} C_VEL
LIN {X 0,Y 420.242,Z 490.555,A -85,B 0,C 180,E1 -10063.744,E2 -10063.744} C_VEL
LIN {X 0,Y 421.734,Z 497.877,A -85,B 0,C 180,E1 -10064.152,E2 -10064.152} C_VEL
LIN {X 0,Y 421.168,Z 510.077,A -85,B 0,C 180,E1 -10064.886,E2 -10064.886} C_VEL
LIN {X 0,Y 420.536,Z 522.081,A -85,B 0,C 180,E1 -10065.821,E2 -10065.821} C_VEL
LIN {X 0,Y 419.871,Z 533.469,A -85,B 0,C 180,E1 -10066.94,E2 -10066.94} C_VEL
LIN {X 0,Y 419.205,Z 543.365,A -85,B 0,C 180,E1 -10068.148,E2 -10068.148} C_VEL
LIN {X 0,Y 418.587,Z 553.011,A -85,B 0,C 180,E1 -10069.601,E2 -10069.601} C_VEL
LIN {X 0,Y 418.094,Z 560.704,A -85,B 0,C 180,E1 -10071.055,E2 -10071.055} C_VEL
LIN {X 0,Y 417.745,Z 566.997,A -85,B 0,C 180,E1 -10072.532,E2 -10072.532} C_VEL
LIN {X 0,Y 417.476,Z 572.561,A -85,B 0,C 180,E1 -10074.203,E2 -10074.203} C_VEL
LIN {X 0,Y 417.333,Z 576.167,A -85,B 0,C 180,E1 -10075.654,E2 -10075.654} C_VEL
LIN {X 0,Y 417.268,Z 578.745,A -85,B 0,C 180,E1 -10077.104,E2 -10077.104} C_VEL
LIN {X 0,Y 417.178,Z 579.92,A -85,B 0,C 180,E1 -10078.069,E2 -10078.069} C_VEL
LIN {X 0,Y 417.117,Z 581.049,A -85,B 0,C 180,E1 -10080,E2 -10080} C_VEL
LIN {X 0,Y 417.182,Z 581.014,A -85,B 0,C 180,E1 -10080.965,E2 -10080.965} C_VEL
LIN {X 0,Y 417.242,Z 580.533,A -85,B 0,C 180,E1 -10081.93,E2 -10081.93} C_VEL
LIN {X 0,Y 417.417,Z 578.375,A -85,B 0,C 180,E1 -10083.861,E2 -10083.861} C_VEL
LIN {X 0,Y 417.462,Z 575.644,A -85,B 0,C 180,E1 -10085.313,E2 -10085.313} C_VEL
LIN {X 0,Y 417.817,Z 571.869,A -85,B 0,C 180,E1 -10086.762,E2 -10086.762} C_VEL
LIN {X 0,Y 418.133,Z 566.977,A -85,B 0,C 180,E1 -10088.214,E2 -10088.214} C_VEL
LIN {X 0,Y 418.652,Z 560.795,A -85,B 0,C 180,E1 -10089.664,E2 -10089.664} C_VEL
LIN {X 0,Y 419.227,Z 553.062,A -85,B 0,C 180,E1 -10091.115,E2 -10091.115} C_VEL
LIN {X 0,Y 419.876,Z 543.49,A -85,B 0,C 180,E1 -10092.568,E2 -10092.568} C_VEL
LIN {X 0,Y 420.846,Z 533.839,A -85,B 0,C 180,E1 -10093.734,E2 -10093.734} C_VEL
LIN {X 0,Y 421.554,Z 522.741,A -85,B 0,C 180,E1 -10094.839,E2 -10094.839} C_VEL
LIN {X 0,Y 422.28,Z 512.072,A -85,B 0,C 180,E1 -10095.691,E2 -10095.691} C_VEL
LIN {X 0,Y 422.949,Z 499.305,A -85,B 0,C 180,E1 -10096.484,E2 -10096.484} C_VEL
LIN {X 0,Y 420.049,Z 488.137,A -85,B 0,C 180,E1 -10097.203,E2 -10097.203} C_VEL
LIN {X 0,Y 417.705,Z 480.801,A -85,B 0,C 180,E1 -10097.661,E2 -10097.661} C_VEL
LIN {X 0,Y 417.802,Z 478.418,A -85,B 0,C 180,E1 -10100.686,E2 -10100.686} C_VEL
LIN {X 0,Y 418.017,Z 476.128,A -85,B 0,C 180,E1 -10103.797,E2 -10103.797} C_VEL
LIN {X 0,Y 418.231,Z 474.005,A -85,B 0,C 180,E1 -10107.048,E2 -10107.048} C_VEL
LIN {X 0,Y 418.477,Z 472.202,A -85,B 0,C 180,E1 -10110.254,E2 -10110.254} C_VEL
LIN {X 0,Y 418.78,Z 470.95,A -85,B 0,C 180,E1 -10112.954,E2 -10112.954} C_VEL
LIN {X 0,Y 419.022,Z 469.994,A -85,B 0,C 180,E1 -10115.947,E2 -10115.947} C_VEL
LIN {X 0,Y 419.081,Z 469.647,A -85,B 0,C 180,E1 -10118.352,E2 -10118.352} C_VEL
LIN {X 0,Y 419.158,Z 469.752,A -85,B 0,C 180,E1 -10121.017,E2 -10121.017} C_VEL
LIN {X 0,Y 419.348,Z 470.531,A -85,B 0,C 180,E1 -10123.891,E2 -10123.891} C_VEL
LIN {X 0,Y 419.619,Z 472.025,A -85,B 0,C 180,E1 -10126.631,E2 -10126.631} C_VEL
LIN {X 0,Y 419.993,Z 474.203,A -85,B 0,C 180,E1 -10129.261,E2 -10129.261} C_VEL
LIN {X 0,Y 420.461,Z 476.971,A -85,B 0,C 180,E1 -10131.796,E2 -10131.796} C_VEL
LIN {X 0,Y 420.497,Z 480.314,A -85,B 0,C 180,E1 -10134.199,E2 -10134.199} C_VEL
LIN {X 0,Y 420.094,Z 484.1,A -85,B 0,C 180,E1 -10136.49,E2 -10136.49} C_VEL
LIN {X 0,Y 419.396,Z 489.309,A -85,B 0,C 180,E1 -10139.263,E2 -10139.263} C_VEL
LIN {X 0,Y 418.728,Z 496.732,A -85,B 0,C 180,E1 -10142.818,E2 -10142.818} C_VEL
LIN {X 0,Y 418.256,Z 503.267,A -85,B 0,C 180,E1 -10145.69,E2 -10145.69} C_VEL
LIN {X 0,Y 417.903,Z 510.731,A -85,B 0,C 180,E1 -10148.803,E2 -10148.803} C_VEL
LIN {X 0,Y 417.572,Z 519.52,A -85,B 0,C 180,E1 -10152.302,E2 -10152.302} C_VEL
LIN {X 0,Y 420.063,Z 533.653,A -85,B 0,C 180,E1 -10152.962,E2 -10152.962} C_VEL
LIN {X 0,Y 421.324,Z 547.931,A -85,B 0,C 180,E1 -10153.775,E2 -10153.775} C_VEL
LIN {X 0,Y 421.473,Z 553.699,A -85,B 0,C 180,E1 -10154.154,E2 -10154.154} C_VEL
LIN {X 0,Y 420.687,Z 565.134,A -85,B 0,C 180,E1 -10154.992,E2 -10154.992} C_VEL
LIN {X 0,Y 419.859,Z 576.214,A -85,B 0,C 180,E1 -10156.002,E2 -10156.002} C_VEL
LIN {X 0,Y 419.054,Z 586.557,A -85,B 0,C 180,E1 -10157.161,E2 -10157.161} C_VEL
LIN {X 0,Y 418.53,Z 595.481,A -85,B 0,C 180,E1 -10158.375,E2 -10158.375} C_VEL
LIN {X 0,Y 417.872,Z 604.273,A -85,B 0,C 180,E1 -10159.828,E2 -10159.828} C_VEL
LIN {X 0,Y 417.535,Z 611.372,A -85,B 0,C 180,E1 -10161.287,E2 -10161.287} C_VEL
LIN {X 0,Y 417.265,Z 617.098,A -85,B 0,C 180,E1 -10162.743,E2 -10162.743} C_VEL
LIN {X 0,Y 417.125,Z 621.609,A -85,B 0,C 180,E1 -10164.198,E2 -10164.198} C_VEL
LIN {X 0,Y 417.151,Z 624.021,A -85,B 0,C 180,E1 -10165.168,E2 -10165.168} C_VEL
LIN {X 0,Y 417.063,Z 625.941,A -85,B 0,C 180,E1 -10166.135,E2 -10166.135} C_VEL
LIN {X 0,Y 417.147,Z 627.413,A -85,B 0,C 180,E1 -10167.103,E2 -10167.103} C_VEL
LIN {X 0,Y 417.133,Z 628.468,A -85,B 0,C 180,E1 -10168.069,E2 -10168.069} C_VEL
LIN {X 0,Y 417.107,Z 629.112,A -85,B 0,C 180,E1 -10169.034,E2 -10169.034} C_VEL
LIN {X 0,Y 417.131,Z 629.3,A -85,B 0,C 180,E1 -10170,E2 -10170} C_VEL
LIN {X 0,Y 417.118,Z 629.068,A -85,B 0,C 180,E1 -10170.965,E2 -10170.965} C_VEL
LIN {X 0,Y 417.132,Z 628.434,A -85,B 0,C 180,E1 -10171.931,E2 -10171.931} C_VEL
LIN {X 0,Y 417.156,Z 627.382,A -85,B 0,C 180,E1 -10172.897,E2 -10172.897} C_VEL
LIN {X 0,Y 417.059,Z 625.846,A -85,B 0,C 180,E1 -10173.865,E2 -10173.865} C_VEL
LIN {X 0,Y 417.166,Z 622.735,A -85,B 0,C 180,E1 -10175.316,E2 -10175.316} C_VEL
LIN {X 0,Y 417.231,Z 618.515,A -85,B 0,C 180,E1 -10176.771,E2 -10176.771} C_VEL
LIN {X 0,Y 417.472,Z 612.068,A -85,B 0,C 180,E1 -10178.471,E2 -10178.471} C_VEL
LIN {X 0,Y 417.823,Z 605.021,A -85,B 0,C 180,E1 -10179.928,E2 -10179.928} C_VEL
LIN {X 0,Y 418.344,Z 596.2,A -85,B 0,C 180,E1 -10181.385,E2 -10181.385} C_VEL
LIN {X 0,Y 418.951,Z 586.224,A -85,B 0,C 180,E1 -10182.719,E2 -10182.719} C_VEL
LIN {X 0,Y 419.703,Z 575.233,A -85,B 0,C 180,E1 -10183.891,E2 -10183.891} C_VEL
LIN {X 0,Y 420.387,Z 563.515,A -85,B 0,C 180,E1 -10184.894,E2 -10184.894} C_VEL
LIN {X 0,Y 421.13,Z 550.991,A -85,B 0,C 180,E1 -10185.721,E2 -10185.721} C_VEL
LIN {X 0,Y 419.705,Z 537.868,A -85,B 0,C 180,E1 -10186.431,E2 -10186.431} C_VEL
LIN {X 0,Y 417.865,Z 524.858,A -85,B 0,C 180,E1 -10186.953,E2 -10186.953} C_VEL
LIN {X 0,Y 417.587,Z 522.68,A -85,B 0,C 180,E1 -10187.022,E2 -10187.022} C_VEL
LIN {X 0,Y 417.913,Z 513.492,A -85,B 0,C 180,E1 -10190.68,E2 -10190.68} C_VEL
LIN {X 0,Y 418.373,Z 504.578,A -85,B 0,C 180,E1 -10194.303,E2 -10194.303} C_VEL
LIN {X 0,Y 418.861,Z 497.534,A -85,B 0,C 180,E1 -10197.217,E2 -10197.217} C_VEL
LIN {X 0,Y 419.3,Z 490.523,A -85,B 0,C 180,E1 -10200.188,E2 -10200.188} C_VEL
LIN {X 0,Y 419.897,Z 483.616,A -85,B 0,C 180,E1 -10203.189,E2 -10203.189} C_VEL
LIN {X 0,Y 420.35,Z 477.74,A -85,B 0,C 180,E1 -10205.816,E2 -10205.816} C_VEL
LIN {X 0,Y 419.733,Z 472.561,A -85,B 0,C 180,E1 -10208.282,E2 -10208.282} C_VEL
LIN {X 0,Y 418.576,Z 466.065,A -85,B 0,C 180,E1 -10211.545,E2 -10211.545} C_VEL
LIN {X 0,Y 418.297,Z 464.382,A -85,B 0,C 180,E1 -10212.452,E2 -10212.452} C_VEL
LIN {X 0,Y 418.285,Z 464.384,A -85,B 0,C 180,E1 -10216.26,E2 -10216.26} C_VEL
LIN {X 0,Y 418.261,Z 464.386,A -85,B 0,C 180,E1 -10219.124,E2 -10219.124} C_VEL
LIN {X 0,Y 418.228,Z 464.388,A -85,B 0,C 180,E1 -10222.167,E2 -10222.167} C_VEL
LIN {X 0,Y 418.266,Z 464.384,A -85,B 0,C 180,E1 -10225.42,E2 -10225.42} C_VEL
LIN {X 0,Y 418.213,Z 464.394,A -85,B 0,C 180,E1 -10228.604,E2 -10228.604} C_VEL
LIN {X 0,Y 418.293,Z 464.381,A -85,B 0,C 180,E1 -10231.937,E2 -10231.937} C_VEL
LIN {X 0,Y 418.291,Z 464.38,A -85,B 0,C 180,E1 -10235.163,E2 -10235.163} C_VEL
LIN {X 0,Y 418.236,Z 464.39,A -85,B 0,C 180,E1 -10238.304,E2 -10238.304} C_VEL
LIN {X 0,Y 418.286,Z 464.38,A -85,B 0,C 180,E1 -10241.383,E2 -10241.383} C_VEL
LIN {X 0,Y 418.305,Z 464.382,A -85,B 0,C 180,E1 -10244.406,E2 -10244.406} C_VEL
LIN {X 0,Y 418.357,Z 464.372,A -85,B 0,C 180,E1 -10247.386,E2 -10247.386} C_VEL
LIN {X 0,Y 418.343,Z 464.376,A -85,B 0,C 180,E1 -10250.329,E2 -10250.329} C_VEL
LIN {X 0,Y 418.496,Z 464.355,A -85,B 0,C 180,E1 -10253.249,E2 -10253.249} C_VEL
LIN {X 0,Y 418.34,Z 464.374,A -85,B 0,C 180,E1 -10255.182,E2 -10255.182} C_VEL
LIN {X 0,Y 418.544,Z 464.349,A -85,B 0,C 180,E1 -10258.076,E2 -10258.076} C_VEL
LIN {X 0,Y 418.675,Z 464.334,A -85,B 0,C 180,E1 -10260,E2 -10260} C_VEL
LIN {X 0,Y 418.511,Z 464.354,A -85,B 0,C 180,E1 -10262.888,E2 -10262.888} C_VEL
LIN {X 0,Y 418.496,Z 464.356,A -85,B 0,C 180,E1 -10266.751,E2 -10266.751} C_VEL
LIN {X 0,Y 418.344,Z 464.374,A -85,B 0,C 180,E1 -10269.672,E2 -10269.672} C_VEL
LIN {X 0,Y 418.349,Z 464.373,A -85,B 0,C 180,E1 -10273.001,E2 -10273.001} C_VEL
LIN {X 0,Y 418.315,Z 464.38,A -85,B 0,C 180,E1 -10276.736,E2 -10276.736} C_VEL
LIN {X 0,Y 418.273,Z 464.382,A -85,B 0,C 180,E1 -10279.791,E2 -10279.791} C_VEL
LIN {X 0,Y 418.24,Z 464.389,A -85,B 0,C 180,E1 -10282.736,E2 -10282.736} C_VEL
LIN {X 0,Y 418.273,Z 464.383,A -85,B 0,C 180,E1 -10285.904,E2 -10285.904} C_VEL
LIN {X 0,Y 418.267,Z 464.383,A -85,B 0,C 180,E1 -10289.162,E2 -10289.162} C_VEL
LIN {X 0,Y 418.26,Z 464.384,A -85,B 0,C 180,E1 -10292.844,E2 -10292.844} C_VEL
LIN {X 0,Y 418.251,Z 464.387,A -85,B 0,C 180,E1 -10296.239,E2 -10296.239} C_VEL
LIN {X 0,Y 418.25,Z 464.385,A -85,B 0,C 180,E1 -10299.683,E2 -10299.683} C_VEL
LIN {X 0,Y 418.235,Z 464.389,A -85,B 0,C 180,E1 -10302.322,E2 -10302.322} C_VEL
LIN {X 0,Y 418.241,Z 464.386,A -85,B 0,C 180,E1 -10305.109,E2 -10305.109} C_VEL
LIN {X 0,Y 418.244,Z 464.386,A -85,B 0,C 180,E1 -10307.767,E2 -10307.767} C_VEL
LIN {X 0,Y 418.26,Z 464.386,A -85,B 0,C 180,E1 -10310.619,E2 -10310.619} C_VEL
LIN {X 0,Y 418.249,Z 464.387,A -85,B 0,C 180,E1 -10313.976,E2 -10313.976} C_VEL
LIN {X 0,Y 418.261,Z 464.384,A -85,B 0,C 180,E1 -10317.156,E2 -10317.156} C_VEL
LIN {X 0,Y 418.272,Z 464.382,A -85,B 0,C 180,E1 -10320.896,E2 -10320.896} C_VEL
LIN {X 0,Y 418.275,Z 464.385,A -85,B 0,C 180,E1 -10324.096,E2 -10324.096} C_VEL
LIN {X 0,Y 418.242,Z 464.386,A -85,B 0,C 180,E1 -10327.264,E2 -10327.264} C_VEL
LIN {X 0,Y 418.287,Z 464.382,A -85,B 0,C 180,E1 -10330.364,E2 -10330.364} C_VEL
LIN {X 0,Y 418.321,Z 464.377,A -85,B 0,C 180,E1 -10333.405,E2 -10333.405} C_VEL
LIN {X 0,Y 418.351,Z 464.371,A -85,B 0,C 180,E1 -10336.999,E2 -10336.999} C_VEL
LIN {X 0,Y 418.345,Z 464.376,A -85,B 0,C 180,E1 -10340.329,E2 -10340.329} C_VEL
LIN {X 0,Y 418.464,Z 464.358,A -85,B 0,C 180,E1 -10343.249,E2 -10343.249} C_VEL
LIN {X 0,Y 418.339,Z 464.373,A -85,B 0,C 180,E1 -10345.182,E2 -10345.182} C_VEL
LIN {X 0,Y 418.548,Z 464.35,A -85,B 0,C 180,E1 -10348.076,E2 -10348.076} C_VEL
LIN {X 0,Y 418.676,Z 464.335,A -85,B 0,C 180,E1 -10350,E2 -10350} C_VEL
LIN {X 0,Y 418.506,Z 464.353,A -85,B 0,C 180,E1 -10352.888,E2 -10352.888} C_VEL
LIN {X 0,Y 418.515,Z 464.354,A -85,B 0,C 180,E1 -10355.783,E2 -10355.783} C_VEL
LIN {X 0,Y 418.4,Z 464.365,A -85,B 0,C 180,E1 -10358.695,E2 -10358.695} C_VEL
LIN {X 0,Y 418.321,Z 464.379,A -85,B 0,C 180,E1 -10361.631,E2 -10361.631} C_VEL
LIN {X 0,Y 418.327,Z 464.376,A -85,B 0,C 180,E1 -10363.332,E2 -10363.332} C_VEL
LIN {X 0,Y 417.634,Z 464.465,A -85,B 0,C 180,E1 -10364.136,E2 -10364.136} C_VEL
LIN {X 0,Y 414.756,Z 464.821,A -85,B 0,C 180,E1 -10365.441,E2 -10365.441} C_VEL
LIN {X 0,Y 412.343,Z 465.121,A -85,B 0,C 180,E1 -10366.495,E2 -10366.495} C_VEL
LIN {X 0,Y 411.321,Z 465.249,A -85,B 0,C 180,E1 -10367.31,E2 -10367.31} C_VEL
LIN {X 0,Y 411.244,Z 465.257,A -85,B 0,C 180,E1 -10367.586,E2 -10367.586} C_VEL
LIN {X 0,Y 411.201,Z 465.263,A -85,B 0,C 180,E1 -10371.034,E2 -10371.034} C_VEL
LIN {X 0,Y 411.232,Z 465.26,A -85,B 0,C 180,E1 -10374.215,E2 -10374.215} C_VEL
LIN {X 0,Y 411.263,Z 465.257,A -85,B 0,C 180,E1 -10377.478,E2 -10377.478} C_VEL
LIN {X 0,Y 411.194,Z 465.263,A -85,B 0,C 180,E1 -10380.847,E2 -10380.847} C_VEL
LIN {X 0,Y 411.21,Z 465.264,A -85,B 0,C 180,E1 -10384.333,E2 -10384.333} C_VEL
LIN {X 0,Y 411.203,Z 465.265,A -85,B 0,C 180,E1 -10387.973,E2 -10387.973} C_VEL
LIN {X 0,Y 411.186,Z 465.266,A -85,B 0,C 180,E1 -10390.504,E2 -10390.504} C_VEL
LIN {X 0,Y 411.177,Z 465.267,A -85,B 0,C 180,E1 -10393.133,E2 -10393.133} C_VEL
LIN {X 0,Y 411.171,Z 465.269,A -85,B 0,C 180,E1 -10395.881,E2 -10395.881} C_VEL
LIN {X 0,Y 411.167,Z 465.267,A -85,B 0,C 180,E1 -10398.772,E2 -10398.772} C_VEL
LIN {X 0,Y 411.206,Z 465.266,A -85,B 0,C 180,E1 -10401.832,E2 -10401.832} C_VEL
LIN {X 0,Y 411.08,Z 465.28,A -85,B 0,C 180,E1 -10405.148,E2 -10405.148} C_VEL
LIN {X 0,Y 410.678,Z 465.33,A -85,B 0,C 180,E1 -10408.833,E2 -10408.833} C_VEL
LIN {X 0,Y 410.451,Z 465.363,A -85,B 0,C 180,E1 -10410.84,E2 -10410.84} C_VEL
LIN {X 0,Y 410.376,Z 467.879,A -85,B 0,C 180,E1 -10413.559,E2 -10413.559} C_VEL
LIN {X 0,Y 410.261,Z 471.165,A -85,B 0,C 180,E1 -10416.796,E2 -10416.796} C_VEL
